LIN {X 0,Y 356.251,Z 232.015,A -85,B 0,C 180,E1 -13438.258,E2 -13438.258} C_VEL
LIN {X 0,Y 354.845,Z 225.287,A -85,B 0,C 180,E1 -13439.964,E2 -13439.964} C_VEL
LIN {X 0,Y 354.802,Z 225.258,A -85,B 0,C 180,E1 -13443.701,E2 -13443.701} C_VEL
LIN {X 0,Y 354.792,Z 225.291,A -85,B 0,C 180,E1 -13446.458,E2 -13446.458} C_VEL
LIN {X 0,Y 354.762,Z 225.285,A -85,B 0,C 180,E1 -13449.411,E2 -13449.411} C_VEL
LIN {X 0,Y 354.779,Z 225.283,A -85,B 0,C 180,E1 -13452.866,E2 -13452.866} C_VEL
LIN {X 0,Y 354.759,Z 225.293,A -85,B 0,C 180,E1 -13456.102,E2 -13456.102} C_VEL
LIN {X 0,Y 354.758,Z 225.282,A -85,B 0,C 180,E1 -13459.175,E2 -13459.175} C_VEL
LIN {X 0,Y 354.793,Z 225.285,A -85,B 0,C 180,E1 -13462.403,E2 -13462.403} C_VEL
LIN {X 0,Y 354.804,Z 225.27,A -85,B 0,C 180,E1 -13464.94,E2 -13464.94} C_VEL
LIN {X 0,Y 354.785,Z 225.285,A -85,B 0,C 180,E1 -13468.404,E2 -13468.404} C_VEL
LIN {X 0,Y 354.788,Z 225.272,A -85,B 0,C 180,E1 -13471.614,E2 -13471.614} C_VEL
LIN {X 0,Y 354.825,Z 225.275,A -85,B 0,C 180,E1 -13475.657,E2 -13475.657} C_VEL
LIN {X 0,Y 354.816,Z 225.265,A -85,B 0,C 180,E1 -13479.113,E2 -13479.113} C_VEL
LIN {X 0,Y 354.869,Z 225.279,A -85,B 0,C 180,E1 -13482.719,E2 -13482.719} C_VEL
LIN {X 0,Y 354.942,Z 225.244,A -85,B 0,C 180,E1 -13486.255,E2 -13486.255} C_VEL
LIN {X 0,Y 354.946,Z 225.269,A -85,B 0,C 180,E1 -13489.735,E2 -13489.735} C_VEL
LIN {X 0,Y 355.073,Z 225.238,A -85,B 0,C 180,E1 -13493.18,E2 -13493.18} C_VEL
LIN {X 0,Y 355.224,Z 225.23,A -85,B 0,C 180,E1 -13497.733,E2 -13497.733} C_VEL
LIN {X 0,Y 355.166,Z 225.228,A -85,B 0,C 180,E1 -13501.134,E2 -13501.134} C_VEL
LIN {X 0,Y 355.221,Z 225.21,A -85,B 0,C 180,E1 -13502.268,E2 -13502.268} C_VEL
LIN {X 0,Y 355.116,Z 225.244,A -85,B 0,C 180,E1 -13506.82,E2 -13506.82} C_VEL
LIN {X 0,Y 354.969,Z 225.243,A -85,B 0,C 180,E1 -13510.265,E2 -13510.265} C_VEL
LIN {X 0,Y 354.935,Z 225.272,A -85,B 0,C 180,E1 -13514.02,E2 -13514.02} C_VEL
LIN {X 0,Y 354.882,Z 225.262,A -85,B 0,C 180,E1 -13518.093,E2 -13518.093} C_VEL
LIN {X 0,Y 354.829,Z 225.279,A -85,B 0,C 180,E1 -13522.107,E2 -13522.107} C_VEL
LIN {X 0,Y 354.893,Z 225.278,A -85,B 0,C 180,E1 -13525.828,E2 -13525.828} C_VEL
LIN {X 0,Y 354.811,Z 225.278,A -85,B 0,C 180,E1 -13529.683,E2 -13529.683} C_VEL
LIN {X 0,Y 354.8,Z 225.28,A -85,B 0,C 180,E1 -13533.703,E2 -13533.703} C_VEL
LIN {X 0,Y 354.794,Z 225.293,A -85,B 0,C 180,E1 -13536.461,E2 -13536.461} C_VEL
LIN {X 0,Y 354.819,Z 225.288,A -85,B 0,C 180,E1 -13539.425,E2 -13539.425} C_VEL
LIN {X 0,Y 354.785,Z 225.29,A -85,B 0,C 180,E1 -13542.869,E2 -13542.869} C_VEL
LIN {X 0,Y 354.766,Z 225.294,A -85,B 0,C 180,E1 -13546.105,E2 -13546.105} C_VEL
LIN {X 0,Y 354.786,Z 225.29,A -85,B 0,C 180,E1 -13549.181,E2 -13549.181} C_VEL
LIN {X 0,Y 354.841,Z 225.283,A -85,B 0,C 180,E1 -13551.977,E2 -13551.977} C_VEL
LIN {X 0,Y 355.818,Z 228.129,A -85,B 0,C 180,E1 -13552.146,E2 -13552.146} C_VEL
LIN {X 0,Y 362.138,Z 240.848,A -85,B 0,C 180,E1 -13552.959,E2 -13552.959} C_VEL
LIN {X 0,Y 365.502,Z 249.264,A -85,B 0,C 180,E1 -13553.412,E2 -13553.412} C_VEL
LIN {X 0,Y 366.502,Z 255.255,A -85,B 0,C 180,E1 -13553.621,E2 -13553.621} C_VEL
LIN {X 0,Y 364.606,Z 337.997,A -85,B 0,C 180,E1 -13555.284,E2 -13555.284} C_VEL
LIN {X 0,Y 364.035,Z 351.449,A -85,B 0,C 180,E1 -13555.767,E2 -13555.767} C_VEL
LIN {X 0,Y 363.357,Z 362.814,A -85,B 0,C 180,E1 -13556.384,E2 -13556.384} C_VEL
LIN {X 0,Y 362.251,Z 374.947,A -85,B 0,C 180,E1 -13557.263,E2 -13557.263} C_VEL
LIN {X 0,Y 361.138,Z 385.976,A -85,B 0,C 180,E1 -13558.304,E2 -13558.304} C_VEL
LIN {X 0,Y 359.839,Z 396.022,A -85,B 0,C 180,E1 -13559.484,E2 -13559.484} C_VEL
LIN {X 0,Y 358.474,Z 406.105,A -85,B 0,C 180,E1 -13560.974,E2 -13560.974} C_VEL
LIN {X 0,Y 357.292,Z 414.918,A -85,B 0,C 180,E1 -13562.599,E2 -13562.599} C_VEL
LIN {X 0,Y 356.138,Z 422.187,A -85,B 0,C 180,E1 -13564.271,E2 -13564.271} C_VEL
LIN {X 0,Y 355.23,Z 428.414,A -85,B 0,C 180,E1 -13566.074,E2 -13566.074} C_VEL
LIN {X 0,Y 354.488,Z 433.26,A -85,B 0,C 180,E1 -13567.873,E2 -13567.873} C_VEL
LIN {X 0,Y 353.956,Z 436.89,A -85,B 0,C 180,E1 -13569.669,E2 -13569.669} C_VEL
LIN {X 0,Y 353.537,Z 439.423,A -85,B 0,C 180,E1 -13571.455,E2 -13571.455} C_VEL
LIN {X 0,Y 353.399,Z 440.56,A -85,B 0,C 180,E1 -13572.665,E2 -13572.665} C_VEL
LIN {X 0,Y 353.286,Z 441.221,A -85,B 0,C 180,E1 -13573.83,E2 -13573.83} C_VEL
LIN {X 0,Y 353.19,Z 441.496,A -85,B 0,C 180,E1 -13575.009,E2 -13575.009} C_VEL
LIN {X 0,Y 353.235,Z 440.909,A -85,B 0,C 180,E1 -13577.14,E2 -13577.14} C_VEL
LIN {X 0,Y 353.276,Z 439.77,A -85,B 0,C 180,E1 -13578.526,E2 -13578.526} C_VEL
LIN {X 0,Y 353.313,Z 438.384,A -85,B 0,C 180,E1 -13579.688,E2 -13579.688} C_VEL
LIN {X 0,Y 353.58,Z 435.443,A -85,B 0,C 180,E1 -13581.428,E2 -13581.428} C_VEL
LIN {X 0,Y 353.899,Z 431.364,A -85,B 0,C 180,E1 -13583.192,E2 -13583.192} C_VEL
LIN {X 0,Y 354.237,Z 426.314,A -85,B 0,C 180,E1 -13584.879,E2 -13584.879} C_VEL
LIN {X 0,Y 354.84,Z 419.838,A -85,B 0,C 180,E1 -13586.595,E2 -13586.595} C_VEL
LIN {X 0,Y 355.605,Z 411.8,A -85,B 0,C 180,E1 -13588.302,E2 -13588.302} C_VEL
LIN {X 0,Y 356.382,Z 403.578,A -85,B 0,C 180,E1 -13589.719,E2 -13589.719} C_VEL
LIN {X 0,Y 357.34,Z 393.444,A -85,B 0,C 180,E1 -13591.128,E2 -13591.128} C_VEL
LIN {X 0,Y 358.376,Z 382.087,A -85,B 0,C 180,E1 -13592.39,E2 -13592.39} C_VEL
LIN {X 0,Y 359.209,Z 370.828,A -85,B 0,C 180,E1 -13593.366,E2 -13593.366} C_VEL
LIN {X 0,Y 359.788,Z 359.435,A -85,B 0,C 180,E1 -13594.132,E2 -13594.132} C_VEL
LIN {X 0,Y 360.335,Z 346.612,A -85,B 0,C 180,E1 -13594.756,E2 -13594.756} C_VEL
LIN {X 0,Y 360.685,Z 334.356,A -85,B 0,C 180,E1 -13595.137,E2 -13595.137} C_VEL
LIN {X 0,Y 361.954,Z 253.14,A -85,B 0,C 180,E1 -13596.743,E2 -13596.743} C_VEL
LIN {X 0,Y 359.063,Z 236.78,A -85,B 0,C 180,E1 -13597.225,E2 -13597.225} C_VEL
LIN {X 0,Y 355.076,Z 225.258,A -85,B 0,C 180,E1 -13597.679,E2 -13597.679} C_VEL
LIN {X 0,Y 354.933,Z 225.27,A -85,B 0,C 180,E1 -13601.515,E2 -13601.515} C_VEL
LIN {X 0,Y 354.233,Z 225.363,A -85,B 0,C 180,E1 -13602.462,E2 -13602.462} C_VEL
LIN {X 0,Y 351.375,Z 225.722,A -85,B 0,C 180,E1 -13604.002,E2 -13604.002} C_VEL
LIN {X 0,Y 348.97,Z 226.024,A -85,B 0,C 180,E1 -13605.248,E2 -13605.248} C_VEL
LIN {X 0,Y 347.931,Z 226.15,A -85,B 0,C 180,E1 -13606.212,E2 -13606.212} C_VEL
LIN {X 0,Y 347.842,Z 226.158,A -85,B 0,C 180,E1 -13606.539,E2 -13606.539} C_VEL
LIN {X 0,Y 347.859,Z 226.152,A -85,B 0,C 180,E1 -13608.861,E2 -13608.861} C_VEL
LIN {X 0,Y 347.762,Z 226.165,A -85,B 0,C 180,E1 -13612.581,E2 -13612.581} C_VEL
LIN {X 0,Y 347.745,Z 226.165,A -85,B 0,C 180,E1 -13615.115,E2 -13615.115} C_VEL
LIN {X 0,Y 347.735,Z 226.169,A -85,B 0,C 180,E1 -13617.702,E2 -13617.702} C_VEL
LIN {X 0,Y 347.744,Z 226.167,A -85,B 0,C 180,E1 -13620.35,E2 -13620.35} C_VEL
LIN {X 0,Y 347.754,Z 226.168,A -85,B 0,C 180,E1 -13624.044,E2 -13624.044} C_VEL
LIN {X 0,Y 347.76,Z 226.166,A -85,B 0,C 180,E1 -13627.322,E2 -13627.322} C_VEL
LIN {X 0,Y 347.702,Z 226.171,A -85,B 0,C 180,E1 -13630.303,E2 -13630.303} C_VEL
LIN {X 0,Y 347.727,Z 226.173,A -85,B 0,C 180,E1 -13633.409,E2 -13633.409} C_VEL
LIN {X 0,Y 347.728,Z 226.168,A -85,B 0,C 180,E1 -13636.687,E2 -13636.687} C_VEL
LIN {X 0,Y 347.707,Z 226.17,A -85,B 0,C 180,E1 -13640.183,E2 -13640.183} C_VEL
LIN {X 0,Y 347.759,Z 226.165,A -85,B 0,C 180,E1 -13642.678,E2 -13642.678} C_VEL
LIN {X 0,Y 347.754,Z 226.164,A -85,B 0,C 180,E1 -13645.957,E2 -13645.957} C_VEL
LIN {X 0,Y 347.735,Z 226.167,A -85,B 0,C 180,E1 -13649.65,E2 -13649.65} C_VEL
LIN {X 0,Y 347.739,Z 226.166,A -85,B 0,C 180,E1 -13653.6,E2 -13653.6} C_VEL
LIN {X 0,Y 347.835,Z 226.225,A -85,B 0,C 180,E1 -13656.362,E2 -13656.362} C_VEL
LIN {X 0,Y 348.763,Z 231.232,A -85,B 0,C 180,E1 -13657.799,E2 -13657.799} C_VEL
LIN {X 0,Y 352.134,Z 244.583,A -85,B 0,C 180,E1 -13658.321,E2 -13658.321} C_VEL
LIN {X 0,Y 354.029,Z 256.193,A -85,B 0,C 180,E1 -13658.724,E2 -13658.724} C_VEL
LIN {X 0,Y 351.664,Z 339.815,A -85,B 0,C 180,E1 -13661.049,E2 -13661.049} C_VEL
LIN {X 0,Y 351.252,Z 352.875,A -85,B 0,C 180,E1 -13661.631,E2 -13661.631} C_VEL
LIN {X 0,Y 350.773,Z 364.722,A -85,B 0,C 180,E1 -13662.359,E2 -13662.359} C_VEL
LIN {X 0,Y 350.003,Z 377.261,A -85,B 0,C 180,E1 -13663.373,E2 -13663.373} C_VEL
LIN {X 0,Y 349.34,Z 388.67,A -85,B 0,C 180,E1 -13664.54,E2 -13664.54} C_VEL
LIN {X 0,Y 348.739,Z 398.714,A -85,B 0,C 180,E1 -13665.812,E2 -13665.812} C_VEL
LIN {X 0,Y 347.973,Z 409.252,A -85,B 0,C 180,E1 -13667.46,E2 -13667.46} C_VEL
LIN {X 0,Y 347.426,Z 416.873,A -85,B 0,C 180,E1 -13668.92,E2 -13668.92} C_VEL
LIN {X 0,Y 346.971,Z 424.322,A -85,B 0,C 180,E1 -13670.674,E2 -13670.674} C_VEL
LIN {X 0,Y 346.661,Z 430.262,A -85,B 0,C 180,E1 -13672.427,E2 -13672.427} C_VEL
LIN {X 0,Y 346.447,Z 434.904,A -85,B 0,C 180,E1 -13674.178,E2 -13674.178} C_VEL
LIN {X 0,Y 346.413,Z 437.37,A -85,B 0,C 180,E1 -13675.345,E2 -13675.345} C_VEL
LIN {X 0,Y 346.311,Z 439.316,A -85,B 0,C 180,E1 -13676.509,E2 -13676.509} C_VEL
LIN {X 0,Y 346.269,Z 440.807,A -85,B 0,C 180,E1 -13677.673,E2 -13677.673} C_VEL
LIN {X 0,Y 346.287,Z 441.878,A -85,B 0,C 180,E1 -13678.837,E2 -13678.837} C_VEL
LIN {X 0,Y 346.363,Z 442.493,A -85,B 0,C 180,E1 -13680,E2 -13680} C_VEL
LIN {X 0,Y 346.448,Z 442.658,A -85,B 0,C 180,E1 -13681.162,E2 -13681.162} C_VEL
LIN {X 0,Y 346.594,Z 442.409,A -85,B 0,C 180,E1 -13682.324,E2 -13682.324} C_VEL
LIN {X 0,Y 346.839,Z 441.74,A -85,B 0,C 180,E1 -13683.485,E2 -13683.485} C_VEL
LIN {X 0,Y 347.127,Z 440.595,A -85,B 0,C 180,E1 -13684.645,E2 -13684.645} C_VEL
LIN {X 0,Y 347.389,Z 439.033,A -85,B 0,C 180,E1 -13685.805,E2 -13685.805} C_VEL
LIN {X 0,Y 347.739,Z 435.862,A -85,B 0,C 180,E1 -13687.548,E2 -13687.548} C_VEL
LIN {X 0,Y 348.683,Z 431.532,A -85,B 0,C 180,E1 -13689.279,E2 -13689.279} C_VEL
LIN {X 0,Y 349.695,Z 426.024,A -85,B 0,C 180,E1 -13691.007,E2 -13691.007} C_VEL
LIN {X 0,Y 350.946,Z 419.105,A -85,B 0,C 180,E1 -13692.726,E2 -13692.726} C_VEL
LIN {X 0,Y 352.377,Z 410.495,A -85,B 0,C 180,E1 -13694.436,E2 -13694.436} C_VEL
LIN {X 0,Y 353.774,Z 401.716,A -85,B 0,C 180,E1 -13695.852,E2 -13695.852} C_VEL
LIN {X 0,Y 355.287,Z 392.173,A -85,B 0,C 180,E1 -13697.112,E2 -13697.112} C_VEL
LIN {X 0,Y 356.87,Z 380.356,A -85,B 0,C 180,E1 -13698.366,E2 -13698.366} C_VEL
LIN {X 0,Y 358.269,Z 368.264,A -85,B 0,C 180,E1 -13699.385,E2 -13699.385} C_VEL
LIN {X 0,Y 359.456,Z 355.545,A -85,B 0,C 180,E1 -13700.199,E2 -13700.199} C_VEL
LIN {X 0,Y 360.443,Z 342.476,A -85,B 0,C 180,E1 -13700.808,E2 -13700.808} C_VEL
LIN {X 0,Y 365.61,Z 264.741,A -85,B 0,C 180,E1 -13703.325,E2 -13703.325} C_VEL
LIN {X 0,Y 360.549,Z 254.309,A -85,B 0,C 180,E1 -13704.498,E2 -13704.498} C_VEL
LIN {X 0,Y 355.99,Z 246.255,A -85,B 0,C 180,E1 -13705.601,E2 -13705.601} C_VEL
LIN {X 0,Y 353.684,Z 242.531,A -85,B 0,C 180,E1 -13706.18,E2 -13706.18} C_VEL
LIN {X 0,Y 351.411,Z 238.71,A -85,B 0,C 180,E1 -13706.823,E2 -13706.823} C_VEL
LIN {X 0,Y 350.201,Z 234.367,A -85,B 0,C 180,E1 -13709.451,E2 -13709.451} C_VEL
LIN {X 0,Y 349.089,Z 230.517,A -85,B 0,C 180,E1 -13712.266,E2 -13712.266} C_VEL
LIN {X 0,Y 348.394,Z 228.278,A -85,B 0,C 180,E1 -13714.391,E2 -13714.391} C_VEL
LIN {X 0,Y 347.767,Z 226.166,A -85,B 0,C 180,E1 -13717.32,E2 -13717.32} C_VEL
LIN {X 0,Y 347.738,Z 226.169,A -85,B 0,C 180,E1 -13720.296,E2 -13720.296} C_VEL
LIN {X 0,Y 347.728,Z 226.171,A -85,B 0,C 180,E1 -13723.407,E2 -13723.407} C_VEL
LIN {X 0,Y 347.752,Z 226.314,A -85,B 0,C 180,E1 -13726.195,E2 -13726.195} C_VEL
LIN {X 0,Y 348.798,Z 229.584,A -85,B 0,C 180,E1 -13729.85,E2 -13729.85} C_VEL
LIN {X 0,Y 350.274,Z 233.844,A -85,B 0,C 180,E1 -13732.99,E2 -13732.99} C_VEL
LIN {X 0,Y 351.793,Z 239.339,A -85,B 0,C 180,E1 -13735.986,E2 -13735.986} C_VEL
LIN {X 0,Y 353.435,Z 245.803,A -85,B 0,C 180,E1 -13738.867,E2 -13738.867} C_VEL
LIN {X 0,Y 354.935,Z 253.192,A -85,B 0,C 180,E1 -13741.625,E2 -13741.625} C_VEL
LIN {X 0,Y 355.556,Z 257.298,A -85,B 0,C 180,E1 -13742.948,E2 -13742.948} C_VEL
LIN {X 0,Y 358.827,Z 269.875,A -85,B 0,C 180,E1 -13744.041,E2 -13744.041} C_VEL
LIN {X 0,Y 361.713,Z 284.255,A -85,B 0,C 180,E1 -13745.081,E2 -13745.081} C_VEL
LIN {X 0,Y 363.46,Z 296.855,A -85,B 0,C 180,E1 -13745.836,E2 -13745.836} C_VEL
LIN {X 0,Y 363.714,Z 302.155,A -85,B 0,C 180,E1 -13746.084,E2 -13746.084} C_VEL
LIN {X 0,Y 359.353,Z 371.007,A -85,B 0,C 180,E1 -13748.298,E2 -13748.298} C_VEL
LIN {X 0,Y 357.977,Z 384.376,A -85,B 0,C 180,E1 -13748.928,E2 -13748.928} C_VEL
LIN {X 0,Y 356.409,Z 397.778,A -85,B 0,C 180,E1 -13749.812,E2 -13749.812} C_VEL
LIN {X 0,Y 354.89,Z 409.166,A -85,B 0,C 180,E1 -13750.777,E2 -13750.777} C_VEL
LIN {X 0,Y 353.186,Z 420.885,A -85,B 0,C 180,E1 -13752.034,E2 -13752.034} C_VEL
LIN {X 0,Y 351.549,Z 431.561,A -85,B 0,C 180,E1 -13753.447,E2 -13753.447} C_VEL
LIN {X 0,Y 350.091,Z 440.352,A -85,B 0,C 180,E1 -13754.871,E2 -13754.871} C_VEL
LIN {X 0,Y 348.869,Z 449.007,A -85,B 0,C 180,E1 -13756.603,E2 -13756.603} C_VEL
LIN {X 0,Y 347.722,Z 456.072,A -85,B 0,C 180,E1 -13758.338,E2 -13758.338} C_VEL
LIN {X 0,Y 347.002,Z 461.759,A -85,B 0,C 180,E1 -13760.086,E2 -13760.086} C_VEL
LIN {X 0,Y 346.55,Z 466.231,A -85,B 0,C 180,E1 -13761.838,E2 -13761.838} C_VEL
LIN {X 0,Y 346.327,Z 468.587,A -85,B 0,C 180,E1 -13763.005,E2 -13763.005} C_VEL
LIN {X 0,Y 346.201,Z 470.469,A -85,B 0,C 180,E1 -13764.173,E2 -13764.173} C_VEL
LIN {X 0,Y 346.171,Z 471.923,A -85,B 0,C 180,E1 -13765.341,E2 -13765.341} C_VEL
LIN {X 0,Y 346.164,Z 472.937,A -85,B 0,C 180,E1 -13766.507,E2 -13766.507} C_VEL
LIN {X 0,Y 346.159,Z 473.475,A -85,B 0,C 180,E1 -13767.672,E2 -13767.672} C_VEL
LIN {X 0,Y 346.29,Z 473.596,A -85,B 0,C 180,E1 -13768.836,E2 -13768.836} C_VEL
LIN {X 0,Y 346.361,Z 473.287,A -85,B 0,C 180,E1 -13769.999,E2 -13769.999} C_VEL
LIN {X 0,Y 346.375,Z 472.501,A -85,B 0,C 180,E1 -13771.161,E2 -13771.161} C_VEL
LIN {X 0,Y 346.207,Z 471.307,A -85,B 0,C 180,E1 -13773.49,E2 -13773.49} C_VEL
LIN {X 0,Y 346.214,Z 470.177,A -85,B 0,C 180,E1 -13774.656,E2 -13774.656} C_VEL
LIN {X 0,Y 346.241,Z 468.394,A -85,B 0,C 180,E1 -13775.955,E2 -13775.955} C_VEL
LIN {X 0,Y 346.508,Z 464.183,A -85,B 0,C 180,E1 -13778.161,E2 -13778.161} C_VEL
LIN {X 0,Y 346.935,Z 459.588,A -85,B 0,C 180,E1 -13779.914,E2 -13779.914} C_VEL
LIN {X 0,Y 347.737,Z 452.634,A -85,B 0,C 180,E1 -13781.955,E2 -13781.955} C_VEL
LIN {X 0,Y 348.863,Z 445.128,A -85,B 0,C 180,E1 -13783.691,E2 -13783.691} C_VEL
LIN {X 0,Y 349.803,Z 437.474,A -85,B 0,C 180,E1 -13785.139,E2 -13785.139} C_VEL
LIN {X 0,Y 351.157,Z 428.129,A -85,B 0,C 180,E1 -13786.569,E2 -13786.569} C_VEL
LIN {X 0,Y 352.603,Z 417.768,A -85,B 0,C 180,E1 -13787.844,E2 -13787.844} C_VEL
LIN {X 0,Y 354.075,Z 406.259,A -85,B 0,C 180,E1 -13788.966,E2 -13788.966} C_VEL
LIN {X 0,Y 355.281,Z 394.013,A -85,B 0,C 180,E1 -13789.875,E2 -13789.875} C_VEL
LIN {X 0,Y 356.446,Z 381.138,A -85,B 0,C 180,E1 -13790.56,E2 -13790.56} C_VEL
LIN {X 0,Y 357.191,Z 368.068,A -85,B 0,C 180,E1 -13791.014,E2 -13791.014} C_VEL
LIN {X 0,Y 358.566,Z 299.255,A -85,B 0,C 180,E1 -13792.452,E2 -13792.452} C_VEL
LIN {X 0,Y 356.048,Z 280.739,A -85,B 0,C 180,E1 -13793.066,E2 -13793.066} C_VEL
LIN {X 0,Y 350.747,Z 250.28,A -85,B 0,C 180,E1 -13794.222,E2 -13794.222} C_VEL
LIN {X 0,Y 351.283,Z 245.173,A -85,B 0,C 180,E1 -13795.395,E2 -13795.395} C_VEL
LIN {X 0,Y 350.496,Z 239.332,A -85,B 0,C 180,E1 -13796.817,E2 -13796.817} C_VEL
LIN {X 0,Y 347.82,Z 226.162,A -85,B 0,C 180,E1 -13800.162,E2 -13800.162} C_VEL
LIN {X 0,Y 347.74,Z 226.141,A -85,B 0,C 180,E1 -13804.463,E2 -13804.463} C_VEL
LIN {X 0,Y 347.757,Z 226.162,A -85,B 0,C 180,E1 -13807.985,E2 -13807.985} C_VEL
LIN {X 0,Y 347.738,Z 226.166,A -85,B 0,C 180,E1 -13811.83,E2 -13811.83} C_VEL
LIN {X 0,Y 347.699,Z 226.171,A -85,B 0,C 180,E1 -13815.026,E2 -13815.026} C_VEL
LIN {X 0,Y 347.734,Z 226.153,A -85,B 0,C 180,E1 -13818.398,E2 -13818.398} C_VEL
LIN {X 0,Y 347.749,Z 226.161,A -85,B 0,C 180,E1 -13822.678,E2 -13822.678} C_VEL
LIN {X 0,Y 347.741,Z 226.162,A -85,B 0,C 180,E1 -13825.955,E2 -13825.955} C_VEL
LIN {X 0,Y 347.732,Z 226.15,A -85,B 0,C 180,E1 -13829.651,E2 -13829.651} C_VEL
LIN {X 0,Y 347.731,Z 226.165,A -85,B 0,C 180,E1 -13833.6,E2 -13833.6} C_VEL
LIN {X 0,Y 347.753,Z 226.156,A -85,B 0,C 180,E1 -13836.159,E2 -13836.159} C_VEL
LIN {X 0,Y 347.789,Z 226.15,A -85,B 0,C 180,E1 -13839.908,E2 -13839.908} C_VEL
LIN {X 0,Y 347.82,Z 226.15,A -85,B 0,C 180,E1 -13843.568,E2 -13843.568} C_VEL
LIN {X 0,Y 347.88,Z 226.13,A -85,B 0,C 180,E1 -13847.16,E2 -13847.16} C_VEL
LIN {X 0,Y 347.926,Z 226.146,A -85,B 0,C 180,E1 -13850.701,E2 -13850.701} C_VEL
LIN {X 0,Y 348.026,Z 226.106,A -85,B 0,C 180,E1 -13854.205,E2 -13854.205} C_VEL
LIN {X 0,Y 348.185,Z 226.106,A -85,B 0,C 180,E1 -13857.687,E2 -13857.687} C_VEL
LIN {X 0,Y 348.134,Z 226.104,A -85,B 0,C 180,E1 -13861.157,E2 -13861.157} C_VEL
LIN {X 0,Y 348.182,Z 226.085,A -85,B 0,C 180,E1 -13862.314,E2 -13862.314} C_VEL
LIN {X 0,Y 348.082,Z 226.12,A -85,B 0,C 180,E1 -13866.958,E2 -13866.958} C_VEL
LIN {X 0,Y 347.92,Z 226.12,A -85,B 0,C 180,E1 -13870.475,E2 -13870.475} C_VEL
LIN {X 0,Y 347.891,Z 226.148,A -85,B 0,C 180,E1 -13874.151,E2 -13874.151} C_VEL
LIN {X 0,Y 347.821,Z 226.143,A -85,B 0,C 180,E1 -13878.26,E2 -13878.26} C_VEL
LIN {X 0,Y 347.783,Z 226.161,A -85,B 0,C 180,E1 -13881.637,E2 -13881.637} C_VEL
LIN {X 0,Y 347.805,Z 226.152,A -85,B 0,C 180,E1 -13885.109,E2 -13885.109} C_VEL
LIN {X 0,Y 347.802,Z 226.157,A -85,B 0,C 180,E1 -13887.695,E2 -13887.695} C_VEL
LIN {X 0,Y 347.743,Z 226.164,A -85,B 0,C 180,E1 -13890.349,E2 -13890.349} C_VEL
LIN {X 0,Y 347.743,Z 226.158,A -85,B 0,C 180,E1 -13894.045,E2 -13894.045} C_VEL
LIN {X 0,Y 347.758,Z 226.165,A -85,B 0,C 180,E1 -13897.322,E2 -13897.322} C_VEL
LIN {X 0,Y 347.729,Z 226.173,A -85,B 0,C 180,E1 -13900.298,E2 -13900.298} C_VEL
LIN {X 0,Y 347.72,Z 226.174,A -85,B 0,C 180,E1 -13903.409,E2 -13903.409} C_VEL
LIN {X 0,Y 347.722,Z 226.172,A -85,B 0,C 180,E1 -13906.688,E2 -13906.688} C_VEL
LIN {X 0,Y 347.745,Z 226.166,A -85,B 0,C 180,E1 -13910.175,E2 -13910.175} C_VEL
LIN {X 0,Y 347.795,Z 226.161,A -85,B 0,C 180,E1 -13911.375,E2 -13911.375} C_VEL
LIN {X 0,Y 348.88,Z 229.117,A -85,B 0,C 180,E1 -13911.557,E2 -13911.557} C_VEL
LIN {X 0,Y 355.974,Z 243.175,A -85,B 0,C 180,E1 -13912.5,E2 -13912.5} C_VEL
LIN {X 0,Y 359.435,Z 251.984,A -85,B 0,C 180,E1 -13912.984,E2 -13912.984} C_VEL
LIN {X 0,Y 360.147,Z 256.344,A -85,B 0,C 180,E1 -13913.139,E2 -13913.139} C_VEL
LIN {X 0,Y 358.158,Z 338.002,A -85,B 0,C 180,E1 -13914.803,E2 -13914.803} C_VEL
LIN {X 0,Y 357.6,Z 351.228,A -85,B 0,C 180,E1 -13915.28,E2 -13915.28} C_VEL
LIN {X 0,Y 356.917,Z 362.189,A -85,B 0,C 180,E1 -13915.869,E2 -13915.869} C_VEL
LIN {X 0,Y 355.784,Z 374.511,A -85,B 0,C 180,E1 -13916.761,E2 -13916.761} C_VEL
LIN {X 0,Y 354.625,Z 385.685,A -85,B 0,C 180,E1 -13917.82,E2 -13917.82} C_VEL
LIN {X 0,Y 353.253,Z 395.856,A -85,B 0,C 180,E1 -13919.019,E2 -13919.019} C_VEL
LIN {X 0,Y 351.934,Z 405.115,A -85,B 0,C 180,E1 -13920.381,E2 -13920.381} C_VEL
LIN {X 0,Y 350.783,Z 413.135,A -85,B 0,C 180,E1 -13921.831,E2 -13921.831} C_VEL
LIN {X 0,Y 349.622,Z 420.41,A -85,B 0,C 180,E1 -13923.433,E2 -13923.433} C_VEL
LIN {X 0,Y 348.634,Z 426.591,A -85,B 0,C 180,E1 -13925.115,E2 -13925.115} C_VEL
LIN {X 0,Y 347.846,Z 431.539,A -85,B 0,C 180,E1 -13926.799,E2 -13926.799} C_VEL
LIN {X 0,Y 347.195,Z 435.707,A -85,B 0,C 180,E1 -13928.633,E2 -13928.633} C_VEL
LIN {X 0,Y 346.833,Z 437.83,A -85,B 0,C 180,E1 -13929.852,E2 -13929.852} C_VEL
LIN {X 0,Y 346.532,Z 439.477,A -85,B 0,C 180,E1 -13931.066,E2 -13931.066} C_VEL
LIN {X 0,Y 346.334,Z 440.868,A -85,B 0,C 180,E1 -13932.508,E2 -13932.508} C_VEL
LIN {X 0,Y 346.11,Z 441.786,A -85,B 0,C 180,E1 -13934.695,E2 -13934.695} C_VEL
LIN {X 0,Y 346.076,Z 441.72,A -85,B 0,C 180,E1 -13935.897,E2 -13935.897} C_VEL
LIN {X 0,Y 346.136,Z 441.22,A -85,B 0,C 180,E1 -13937.096,E2 -13937.096} C_VEL
LIN {X 0,Y 346.166,Z 440.291,A -85,B 0,C 180,E1 -13938.288,E2 -13938.288} C_VEL
LIN {X 0,Y 346.203,Z 438.968,A -85,B 0,C 180,E1 -13939.474,E2 -13939.474} C_VEL
LIN {X 0,Y 346.454,Z 436.147,A -85,B 0,C 180,E1 -13941.25,E2 -13941.25} C_VEL
LIN {X 0,Y 346.819,Z 431.855,A -85,B 0,C 180,E1 -13943.195,E2 -13943.195} C_VEL
LIN {X 0,Y 347.129,Z 427.318,A -85,B 0,C 180,E1 -13944.774,E2 -13944.774} C_VEL
LIN {X 0,Y 347.739,Z 421.016,A -85,B 0,C 180,E1 -13946.525,E2 -13946.525} C_VEL
LIN {X 0,Y 348.485,Z 413.157,A -85,B 0,C 180,E1 -13948.268,E2 -13948.268} C_VEL
LIN {X 0,Y 349.287,Z 405.14,A -85,B 0,C 180,E1 -13949.713,E2 -13949.713} C_VEL
LIN {X 0,Y 350.251,Z 395.376,A -85,B 0,C 180,E1 -13951.151,E2 -13951.151} C_VEL
LIN {X 0,Y 351.314,Z 384.221,A -85,B 0,C 180,E1 -13952.452,E2 -13952.452} C_VEL
LIN {X 0,Y 352.283,Z 372.062,A -85,B 0,C 180,E1 -13953.566,E2 -13953.566} C_VEL
LIN {X 0,Y 352.928,Z 359.939,A -85,B 0,C 180,E1 -13954.405,E2 -13954.405} C_VEL
LIN {X 0,Y 353.517,Z 346.676,A -85,B 0,C 180,E1 -13955.062,E2 -13955.062} C_VEL
LIN {X 0,Y 353.863,Z 334.204,A -85,B 0,C 180,E1 -13955.45,E2 -13955.45} C_VEL
LIN {X 0,Y 355.189,Z 254.031,A -85,B 0,C 180,E1 -13957.064,E2 -13957.064} C_VEL
LIN {X 0,Y 352.559,Z 238.973,A -85,B 0,C 180,E1 -13957.517,E2 -13957.517} C_VEL
LIN {X 0,Y 348.023,Z 226.135,A -85,B 0,C 180,E1 -13958.049,E2 -13958.049} C_VEL
LIN {X 0,Y 347.889,Z 226.147,A -85,B 0,C 180,E1 -13961.656,E2 -13961.656} C_VEL
LIN {X 0,Y 347.872,Z 226.15,A -85,B 0,C 180,E1 -13965.228,E2 -13965.228} C_VEL
LIN {X 0,Y 347.842,Z 226.158,A -85,B 0,C 180,E1 -13966.539,E2 -13966.539} C_VEL
LIN {X 0,Y 347.148,Z 226.241,A -85,B 0,C 180,E1 -13967.505,E2 -13967.505} C_VEL
LIN {X 0,Y 344.244,Z 226.602,A -85,B 0,C 180,E1 -13969.075,E2 -13969.075} C_VEL
LIN {X 0,Y 341.811,Z 226.91,A -85,B 0,C 180,E1 -13970.346,E2 -13970.346} C_VEL
LIN {X 0,Y 340.792,Z 227.032,A -85,B 0,C 180,E1 -13971.331,E2 -13971.331} C_VEL
LIN {X 0,Y 340.723,Z 227.041,A -85,B 0,C 180,E1 -13971.664,E2 -13971.664} C_VEL
LIN {X 0,Y 340.714,Z 227.042,A -85,B 0,C 180,E1 -13974.823,E2 -13974.823} C_VEL
LIN {X 0,Y 340.685,Z 227.047,A -85,B 0,C 180,E1 -13978.326,E2 -13978.326} C_VEL
LIN {X 0,Y 340.7,Z 227.043,A -85,B 0,C 180,E1 -13981.046,E2 -13981.046} C_VEL
LIN {X 0,Y 340.722,Z 227.042,A -85,B 0,C 180,E1 -13985.28,E2 -13985.28} C_VEL
LIN {X 0,Y 340.699,Z 227.043,A -85,B 0,C 180,E1 -13988.383,E2 -13988.383} C_VEL
LIN {X 0,Y 340.696,Z 227.044,A -85,B 0,C 180,E1 -13992.044,E2 -13992.044} C_VEL
LIN {X 0,Y 340.655,Z 227.048,A -85,B 0,C 180,E1 -13996.228,E2 -13996.228} C_VEL
LIN {X 0,Y 340.674,Z 227.047,A -85,B 0,C 180,E1 -13998.688,E2 -13998.688} C_VEL
LIN {X 0,Y 340.723,Z 227.041,A -85,B 0,C 180,E1 -14001.771,E2 -14001.771} C_VEL
LIN {X 0,Y 340.728,Z 227.041,A -85,B 0,C 180,E1 -14005.596,E2 -14005.596} C_VEL
LIN {X 0,Y 340.688,Z 227.05,A -85,B 0,C 180,E1 -14008.954,E2 -14008.954} C_VEL
LIN {X 0,Y 340.692,Z 227.046,A -85,B 0,C 180,E1 -14012.505,E2 -14012.505} C_VEL
LIN {X 0,Y 340.784,Z 227.049,A -85,B 0,C 180,E1 -14016.206,E2 -14016.206} C_VEL
LIN {X 0,Y 341.6,Z 231.537,A -85,B 0,C 180,E1 -14017.512,E2 -14017.512} C_VEL
LIN {X 0,Y 345.32,Z 245.986,A -85,B 0,C 180,E1 -14018.096,E2 -14018.096} C_VEL
LIN {X 0,Y 347.119,Z 256.377,A -85,B 0,C 180,E1 -14018.472,E2 -14018.472} C_VEL
LIN {X 0,Y 344.644,Z 340.237,A -85,B 0,C 180,E1 -14020.88,E2 -14020.88} C_VEL
LIN {X 0,Y 344.191,Z 354.626,A -85,B 0,C 180,E1 -14021.549,E2 -14021.549} C_VEL
LIN {X 0,Y 343.598,Z 367.998,A -85,B 0,C 180,E1 -14022.44,E2 -14022.44} C_VEL
LIN {X 0,Y 342.83,Z 379.972,A -85,B 0,C 180,E1 -14023.474,E2 -14023.474} C_VEL
LIN {X 0,Y 342.061,Z 391.134,A -85,B 0,C 180,E1 -14024.698,E2 -14024.698} C_VEL
LIN {X 0,Y 341.557,Z 400.868,A -85,B 0,C 180,E1 -14026.008,E2 -14026.008} C_VEL
LIN {X 0,Y 340.845,Z 410.007,A -85,B 0,C 180,E1 -14027.496,E2 -14027.496} C_VEL
LIN {X 0,Y 340.245,Z 418.883,A -85,B 0,C 180,E1 -14029.286,E2 -14029.286} C_VEL
LIN {X 0,Y 339.795,Z 426.015,A -85,B 0,C 180,E1 -14031.076,E2 -14031.076} C_VEL
LIN {X 0,Y 339.485,Z 431.702,A -85,B 0,C 180,E1 -14032.864,E2 -14032.864} C_VEL
LIN {X 0,Y 339.326,Z 436.112,A -85,B 0,C 180,E1 -14034.652,E2 -14034.652} C_VEL
LIN {X 0,Y 339.234,Z 439.371,A -85,B 0,C 180,E1 -14036.436,E2 -14036.436} C_VEL
LIN {X 0,Y 339.176,Z 440.937,A -85,B 0,C 180,E1 -14037.625,E2 -14037.625} C_VEL
LIN {X 0,Y 339.19,Z 442.074,A -85,B 0,C 180,E1 -14038.812,E2 -14038.812} C_VEL
LIN {X 0,Y 339.268,Z 442.796,A -85,B 0,C 180,E1 -14040,E2 -14040} C_VEL
LIN {X 0,Y 339.389,Z 443.05,A -85,B 0,C 180,E1 -14041.186,E2 -14041.186} C_VEL
LIN {X 0,Y 339.543,Z 442.868,A -85,B 0,C 180,E1 -14042.372,E2 -14042.372} C_VEL
LIN {X 0,Y 339.799,Z 442.274,A -85,B 0,C 180,E1 -14043.557,E2 -14043.557} C_VEL
LIN {X 0,Y 340.1,Z 441.253,A -85,B 0,C 180,E1 -14044.741,E2 -14044.741} C_VEL
LIN {X 0,Y 340.369,Z 439.762,A -85,B 0,C 180,E1 -14045.926,E2 -14045.926} C_VEL
LIN {X 0,Y 340.756,Z 436.736,A -85,B 0,C 180,E1 -14047.704,E2 -14047.704} C_VEL
LIN {X 0,Y 341.753,Z 432.563,A -85,B 0,C 180,E1 -14049.469,E2 -14049.469} C_VEL
LIN {X 0,Y 343.063,Z 426.214,A -85,B 0,C 180,E1 -14051.521,E2 -14051.521} C_VEL
LIN {X 0,Y 344.385,Z 419.252,A -85,B 0,C 180,E1 -14053.272,E2 -14053.272} C_VEL
LIN {X 0,Y 345.958,Z 410.61,A -85,B 0,C 180,E1 -14055.011,E2 -14055.011} C_VEL
LIN {X 0,Y 347.687,Z 400.817,A -85,B 0,C 180,E1 -14056.59,E2 -14056.59} C_VEL
LIN {X 0,Y 349.471,Z 389.781,A -85,B 0,C 180,E1 -14058.011,E2 -14058.011} C_VEL
LIN {X 0,Y 350.97,Z 379.08,A -85,B 0,C 180,E1 -14059.125,E2 -14059.125} C_VEL
LIN {X 0,Y 352.486,Z 366.829,A -85,B 0,C 180,E1 -14060.128,E2 -14060.128} C_VEL
LIN {X 0,Y 353.76,Z 353.226,A -85,B 0,C 180,E1 -14060.983,E2 -14060.983} C_VEL
LIN {X 0,Y 354.887,Z 337.752,A -85,B 0,C 180,E1 -14061.643,E2 -14061.643} C_VEL
LIN {X 0,Y 360.039,Z 267.819,A -85,B 0,C 180,E1 -14063.955,E2 -14063.955} C_VEL
LIN {X 0,Y 359.7,Z 266.468,A -85,B 0,C 180,E1 -14064.066,E2 -14064.066} C_VEL
LIN {X 0,Y 354.327,Z 255.635,A -85,B 0,C 180,E1 -14065.405,E2 -14065.405} C_VEL
LIN {X 0,Y 349.549,Z 247.582,A -85,B 0,C 180,E1 -14066.657,E2 -14066.657} C_VEL
LIN {X 0,Y 346.812,Z 243.405,A -85,B 0,C 180,E1 -14067.412,E2 -14067.412} C_VEL
LIN {X 0,Y 344.489,Z 239.643,A -85,B 0,C 180,E1 -14068.115,E2 -14068.115} C_VEL
LIN {X 0,Y 343.375,Z 235.771,A -85,B 0,C 180,E1 -14070.776,E2 -14070.776} C_VEL
LIN {X 0,Y 342.404,Z 232.42,A -85,B 0,C 180,E1 -14073.655,E2 -14073.655} C_VEL
LIN {X 0,Y 341.674,Z 230.014,A -85,B 0,C 180,E1 -14076.657,E2 -14076.657} C_VEL
LIN {X 0,Y 341.159,Z 228.768,A -85,B 0,C 180,E1 -14079.688,E2 -14079.688} C_VEL
LIN {X 0,Y 341.091,Z 228.68,A -85,B 0,C 180,E1 -14082.839,E2 -14082.839} C_VEL
LIN {X 0,Y 341.647,Z 229.85,A -85,B 0,C 180,E1 -14086.053,E2 -14086.053} C_VEL
LIN {X 0,Y 342.47,Z 232.706,A -85,B 0,C 180,E1 -14089.402,E2 -14089.402} C_VEL
LIN {X 0,Y 343.978,Z 237.078,A -85,B 0,C 180,E1 -14092.828,E2 -14092.828} C_VEL
LIN {X 0,Y 345.531,Z 242.679,A -85,B 0,C 180,E1 -14095.989,E2 -14095.989} C_VEL
LIN {X 0,Y 347.218,Z 249.706,A -85,B 0,C 180,E1 -14099.158,E2 -14099.158} C_VEL
LIN {X 0,Y 348.502,Z 256.425,A -85,B 0,C 180,E1 -14101.693,E2 -14101.693} C_VEL
LIN {X 0,Y 350.746,Z 261.246,A -85,B 0,C 180,E1 -14102.347,E2 -14102.347} C_VEL
LIN {X 0,Y 353.132,Z 270.252,A -85,B 0,C 180,E1 -14103.193,E2 -14103.193} C_VEL
LIN {X 0,Y 355.865,Z 283.758,A -85,B 0,C 180,E1 -14104.247,E2 -14104.247} C_VEL
LIN {X 0,Y 357.73,Z 296.729,A -85,B 0,C 180,E1 -14105.09,E2 -14105.09} C_VEL
LIN {X 0,Y 358.082,Z 303.505,A -85,B 0,C 180,E1 -14105.43,E2 -14105.43} C_VEL
LIN {X 0,Y 353.463,Z 370.44,A -85,B 0,C 180,E1 -14107.649,E2 -14107.649} C_VEL
LIN {X 0,Y 351.955,Z 384.282,A -85,B 0,C 180,E1 -14108.319,E2 -14108.319} C_VEL
LIN {X 0,Y 350.146,Z 398.443,A -85,B 0,C 180,E1 -14109.281,E2 -14109.281} C_VEL
LIN {X 0,Y 348.307,Z 410.903,A -85,B 0,C 180,E1 -14110.399,E2 -14110.399} C_VEL
LIN {X 0,Y 346.332,Z 423.358,A -85,B 0,C 180,E1 -14111.819,E2 -14111.819} C_VEL
LIN {X 0,Y 344.506,Z 434.331,A -85,B 0,C 180,E1 -14113.404,E2 -14113.404} C_VEL
LIN {X 0,Y 343.024,Z 442.595,A -85,B 0,C 180,E1 -14114.856,E2 -14114.856} C_VEL
LIN {X 0,Y 341.743,Z 450.759,A -85,B 0,C 180,E1 -14116.622,E2 -14116.622} C_VEL
LIN {X 0,Y 340.758,Z 456.402,A -85,B 0,C 180,E1 -14118.096,E2 -14118.096} C_VEL
LIN {X 0,Y 339.999,Z 461.92,A -85,B 0,C 180,E1 -14119.879,E2 -14119.879} C_VEL
LIN {X 0,Y 339.512,Z 466.26,A -85,B 0,C 180,E1 -14121.667,E2 -14121.667} C_VEL
LIN {X 0,Y 339.258,Z 468.523,A -85,B 0,C 180,E1 -14122.859,E2 -14122.859} C_VEL
LIN {X 0,Y 339.133,Z 470.437,A -85,B 0,C 180,E1 -14124.113,E2 -14124.113} C_VEL
LIN {X 0,Y 339.072,Z 471.742,A -85,B 0,C 180,E1 -14125.243,E2 -14125.243} C_VEL
LIN {X 0,Y 339.086,Z 472.655,A -85,B 0,C 180,E1 -14126.434,E2 -14126.434} C_VEL
LIN {X 0,Y 339.068,Z 473.14,A -85,B 0,C 180,E1 -14127.623,E2 -14127.623} C_VEL
LIN {X 0,Y 339.194,Z 473.209,A -85,B 0,C 180,E1 -14128.811,E2 -14128.811} C_VEL
LIN {X 0,Y 339.3,Z 472.819,A -85,B 0,C 180,E1 -14129.999,E2 -14129.999} C_VEL
LIN {X 0,Y 339.294,Z 472.054,A -85,B 0,C 180,E1 -14131.186,E2 -14131.186} C_VEL
LIN {X 0,Y 339.128,Z 471.044,A -85,B 0,C 180,E1 -14133.563,E2 -14133.563} C_VEL
LIN {X 0,Y 339.114,Z 469.949,A -85,B 0,C 180,E1 -14134.754,E2 -14134.754} C_VEL
LIN {X 0,Y 339.169,Z 468.398,A -85,B 0,C 180,E1 -14135.946,E2 -14135.946} C_VEL
LIN {X 0,Y 339.338,Z 465.286,A -85,B 0,C 180,E1 -14137.735,E2 -14137.735} C_VEL
LIN {X 0,Y 339.718,Z 461.118,A -85,B 0,C 180,E1 -14139.525,E2 -14139.525} C_VEL
LIN {X 0,Y 340.453,Z 454.762,A -85,B 0,C 180,E1 -14141.61,E2 -14141.61} C_VEL
LIN {X 0,Y 341.572,Z 447.857,A -85,B 0,C 180,E1 -14143.382,E2 -14143.382} C_VEL
LIN {X 0,Y 342.726,Z 439.218,A -85,B 0,C 180,E1 -14145.155,E2 -14145.155} C_VEL
LIN {X 0,Y 344.034,Z 430.373,A -85,B 0,C 180,E1 -14146.617,E2 -14146.617} C_VEL
LIN {X 0,Y 345.562,Z 420.653,A -85,B 0,C 180,E1 -14147.914,E2 -14147.914} C_VEL
LIN {X 0,Y 346.989,Z 409.948,A -85,B 0,C 180,E1 -14149.061,E2 -14149.061} C_VEL
LIN {X 0,Y 348.334,Z 397.962,A -85,B 0,C 180,E1 -14150.058,E2 -14150.058} C_VEL
LIN {X 0,Y 349.617,Z 385.43,A -85,B 0,C 180,E1 -14150.826,E2 -14150.826} C_VEL
LIN {X 0,Y 350.604,Z 372.2,A -85,B 0,C 180,E1 -14151.369,E2 -14151.369} C_VEL
LIN {X 0,Y 351.072,Z 355.495,A -85,B 0,C 180,E1 -14151.78,E2 -14151.78} C_VEL
LIN {X 0,Y 352.176,Z 299.865,A -85,B 0,C 180,E1 -14152.951,E2 -14152.951} C_VEL
LIN {X 0,Y 349.492,Z 280.321,A -85,B 0,C 180,E1 -14153.622,E2 -14153.622} C_VEL
LIN {X 0,Y 343.988,Z 248.665,A -85,B 0,C 180,E1 -14154.88,E2 -14154.88} C_VEL
LIN {X 0,Y 344.26,Z 245.227,A -85,B 0,C 180,E1 -14155.693,E2 -14155.693} C_VEL
LIN {X 0,Y 342.468,Z 235.404,A -85,B 0,C 180,E1 -14158.162,E2 -14158.162} C_VEL
LIN {X 0,Y 340.752,Z 227.042,A -85,B 0,C 180,E1 -14160.365,E2 -14160.365} C_VEL
LIN {X 0,Y 340.718,Z 227.014,A -85,B 0,C 180,E1 -14164.403,E2 -14164.403} C_VEL
LIN {X 0,Y 340.713,Z 227.037,A -85,B 0,C 180,E1 -14168.228,E2 -14168.228} C_VEL
LIN {X 0,Y 340.687,Z 227.043,A -85,B 0,C 180,E1 -14172.043,E2 -14172.043} C_VEL
LIN {X 0,Y 340.645,Z 227.051,A -85,B 0,C 180,E1 -14176.226,E2 -14176.226} C_VEL
LIN {X 0,Y 340.663,Z 227.034,A -85,B 0,C 180,E1 -14178.687,E2 -14178.687} C_VEL
LIN {X 0,Y 340.711,Z 227.041,A -85,B 0,C 180,E1 -14181.77,E2 -14181.77} C_VEL
LIN {X 0,Y 340.715,Z 227.032,A -85,B 0,C 180,E1 -14185.595,E2 -14185.595} C_VEL
LIN {X 0,Y 340.686,Z 227.035,A -85,B 0,C 180,E1 -14188.954,E2 -14188.954} C_VEL
LIN {X 0,Y 340.703,Z 227.036,A -85,B 0,C 180,E1 -14193.011,E2 -14193.011} C_VEL
LIN {X 0,Y 340.73,Z 227.031,A -85,B 0,C 180,E1 -14195.637,E2 -14195.637} C_VEL
LIN {X 0,Y 340.719,Z 227.025,A -85,B 0,C 180,E1 -14199.473,E2 -14199.473} C_VEL
LIN {X 0,Y 340.783,Z 227.031,A -85,B 0,C 180,E1 -14201.98,E2 -14201.98} C_VEL
LIN {X 0,Y 340.844,Z 226.999,A -85,B 0,C 180,E1 -14205.716,E2 -14205.716} C_VEL
LIN {X 0,Y 340.838,Z 227.027,A -85,B 0,C 180,E1 -14209.305,E2 -14209.305} C_VEL
LIN {X 0,Y 340.988,Z 226.994,A -85,B 0,C 180,E1 -14212.897,E2 -14212.897} C_VEL
LIN {X 0,Y 340.809,Z 227.006,A -85,B 0,C 180,E1 -14215.269,E2 -14215.269} C_VEL
LIN {X 0,Y 341.146,Z 226.983,A -85,B 0,C 180,E1 -14217.639,E2 -14217.639} C_VEL
LIN {X 0,Y 341.103,Z 226.98,A -85,B 0,C 180,E1 -14221.181,E2 -14221.181} C_VEL
LIN {X 0,Y 341.12,Z 226.964,A -85,B 0,C 180,E1 -14222.362,E2 -14222.362} C_VEL
LIN {X 0,Y 341.05,Z 226.996,A -85,B 0,C 180,E1 -14227.103,E2 -14227.103} C_VEL
LIN {X 0,Y 340.862,Z 226.999,A -85,B 0,C 180,E1 -14230.694,E2 -14230.694} C_VEL
LIN {X 0,Y 340.855,Z 227.023,A -85,B 0,C 180,E1 -14234.326,E2 -14234.326} C_VEL
LIN {X 0,Y 340.778,Z 227.022,A -85,B 0,C 180,E1 -14238.441,E2 -14238.441} C_VEL
LIN {X 0,Y 340.747,Z 227.035,A -85,B 0,C 180,E1 -14241.858,E2 -14241.858} C_VEL
LIN {X 0,Y 340.766,Z 227.034,A -85,B 0,C 180,E1 -14245.665,E2 -14245.665} C_VEL
LIN {X 0,Y 340.722,Z 227.035,A -85,B 0,C 180,E1 -14248.322,E2 -14248.322} C_VEL
LIN {X 0,Y 340.692,Z 227.045,A -85,B 0,C 180,E1 -14251.046,E2 -14251.046} C_VEL
LIN {X 0,Y 340.713,Z 227.041,A -85,B 0,C 180,E1 -14255.28,E2 -14255.28} C_VEL
LIN {X 0,Y 340.706,Z 227.038,A -85,B 0,C 180,E1 -14258.387,E2 -14258.387} C_VEL
LIN {X 0,Y 340.695,Z 227.04,A -85,B 0,C 180,E1 -14262.047,E2 -14262.047} C_VEL
LIN {X 0,Y 340.649,Z 227.053,A -85,B 0,C 180,E1 -14266.228,E2 -14266.228} C_VEL
LIN {X 0,Y 340.686,Z 227.044,A -85,B 0,C 180,E1 -14269.754,E2 -14269.754} C_VEL
LIN {X 0,Y 340.727,Z 227.045,A -85,B 0,C 180,E1 -14270.736,E2 -14270.736} C_VEL
LIN {X 0,Y 341.821,Z 230.007,A -85,B 0,C 180,E1 -14270.922,E2 -14270.922} C_VEL
LIN {X 0,Y 349.737,Z 245.378,A -85,B 0,C 180,E1 -14272.01,E2 -14272.01} C_VEL
LIN {X 0,Y 353.365,Z 254.4,A -85,B 0,C 180,E1 -14272.532,E2 -14272.532} C_VEL
LIN {X 0,Y 353.805,Z 257.888,A -85,B 0,C 180,E1 -14272.649,E2 -14272.649} C_VEL
LIN {X 0,Y 351.747,Z 338.734,A -85,B 0,C 180,E1 -14274.328,E2 -14274.328} C_VEL
LIN {X 0,Y 351.144,Z 351.956,A -85,B 0,C 180,E1 -14274.818,E2 -14274.818} C_VEL
LIN {X 0,Y 350.367,Z 363.773,A -85,B 0,C 180,E1 -14275.483,E2 -14275.483} C_VEL
LIN {X 0,Y 349.157,Z 375.854,A -85,B 0,C 180,E1 -14276.392,E2 -14276.392} C_VEL
LIN {X 0,Y 347.951,Z 386.836,A -85,B 0,C 180,E1 -14277.469,E2 -14277.469} C_VEL
LIN {X 0,Y 346.547,Z 396.597,A -85,B 0,C 180,E1 -14278.657,E2 -14278.657} C_VEL
LIN {X 0,Y 345.162,Z 405.96,A -85,B 0,C 180,E1 -14280.077,E2 -14280.077} C_VEL
LIN {X 0,Y 343.884,Z 414.21,A -85,B 0,C 180,E1 -14281.617,E2 -14281.617} C_VEL
LIN {X 0,Y 342.503,Z 422.323,A -85,B 0,C 180,E1 -14283.495,E2 -14283.495} C_VEL
LIN {X 0,Y 341.502,Z 428.289,A -85,B 0,C 180,E1 -14285.248,E2 -14285.248} C_VEL
LIN {X 0,Y 340.731,Z 432.855,A -85,B 0,C 180,E1 -14286.929,E2 -14286.929} C_VEL
LIN {X 0,Y 340.221,Z 435.962,A -85,B 0,C 180,E1 -14288.37,E2 -14288.37} C_VEL
LIN {X 0,Y 339.878,Z 437.817,A -85,B 0,C 180,E1 -14289.421,E2 -14289.421} C_VEL
LIN {X 0,Y 339.531,Z 439.532,A -85,B 0,C 180,E1 -14290.661,E2 -14290.661} C_VEL
LIN {X 0,Y 339.264,Z 441.181,A -85,B 0,C 180,E1 -14292.349,E2 -14292.349} C_VEL
LIN {X 0,Y 339.038,Z 442.077,A -85,B 0,C 180,E1 -14294.368,E2 -14294.368} C_VEL
LIN {X 0,Y 338.982,Z 442.068,A -85,B 0,C 180,E1 -14295.595,E2 -14295.595} C_VEL
LIN {X 0,Y 339.03,Z 441.574,A -85,B 0,C 180,E1 -14296.984,E2 -14296.984} C_VEL
LIN {X 0,Y 339.103,Z 439.545,A -85,B 0,C 180,E1 -14299.251,E2 -14299.251} C_VEL
LIN {X 0,Y 339.346,Z 436.843,A -85,B 0,C 180,E1 -14301.066,E2 -14301.066} C_VEL
LIN {X 0,Y 339.733,Z 432.32,A -85,B 0,C 180,E1 -14303.206,E2 -14303.206} C_VEL
LIN {X 0,Y 340.027,Z 428.271,A -85,B 0,C 180,E1 -14304.665,E2 -14304.665} C_VEL
LIN {X 0,Y 340.641,Z 422.156,A -85,B 0,C 180,E1 -14306.453,E2 -14306.453} C_VEL
LIN {X 0,Y 341.376,Z 414.509,A -85,B 0,C 180,E1 -14308.232,E2 -14308.232} C_VEL
LIN {X 0,Y 342.356,Z 404.953,A -85,B 0,C 180,E1 -14310.001,E2 -14310.001} C_VEL
LIN {X 0,Y 343.36,Z 395.035,A -85,B 0,C 180,E1 -14311.467,E2 -14311.467} C_VEL
LIN {X 0,Y 344.506,Z 383.454,A -85,B 0,C 180,E1 -14312.822,E2 -14312.822} C_VEL
LIN {X 0,Y 345.352,Z 372.801,A -85,B 0,C 180,E1 -14313.809,E2 -14313.809} C_VEL
LIN {X 0,Y 346.039,Z 360.857,A -85,B 0,C 180,E1 -14314.661,E2 -14314.661} C_VEL
LIN {X 0,Y 346.615,Z 347.523,A -85,B 0,C 180,E1 -14315.346,E2 -14315.346} C_VEL
LIN {X 0,Y 347.032,Z 335.458,A -85,B 0,C 180,E1 -14315.74,E2 -14315.74} C_VEL
LIN {X 0,Y 348.436,Z 254.885,A -85,B 0,C 180,E1 -14317.394,E2 -14317.394} C_VEL
LIN {X 0,Y 345.949,Z 240.825,A -85,B 0,C 180,E1 -14317.828,E2 -14317.828} C_VEL
LIN {X 0,Y 341.004,Z 227.145,A -85,B 0,C 180,E1 -14318.398,E2 -14318.398} C_VEL
LIN {X 0,Y 340.855,Z 227.024,A -85,B 0,C 180,E1 -14321.9,E2 -14321.9} C_VEL
LIN {X 0,Y 340.826,Z 227.027,A -85,B 0,C 180,E1 -14325.551,E2 -14325.551} C_VEL
LIN {X 0,Y 340.844,Z 227.029,A -85,B 0,C 180,E1 -14328.467,E2 -14328.467} C_VEL
LIN {X 0,Y 340.723,Z 227.041,A -85,B 0,C 180,E1 -14331.664,E2 -14331.664} C_VEL
LIN {X 0,Y 340.081,Z 227.125,A -85,B 0,C 180,E1 -14332.652,E2 -14332.652} C_VEL
LIN {X 0,Y 337.199,Z 227.486,A -85,B 0,C 180,E1 -14334.257,E2 -14334.257} C_VEL
LIN {X 0,Y 334.745,Z 227.788,A -85,B 0,C 180,E1 -14335.557,E2 -14335.557} C_VEL
LIN {X 0,Y 333.704,Z 227.916,A -85,B 0,C 180,E1 -14336.564,E2 -14336.564} C_VEL
LIN {X 0,Y 333.627,Z 227.924,A -85,B 0,C 180,E1 -14336.905,E2 -14336.905} C_VEL
LIN {X 0,Y 333.663,Z 227.921,A -85,B 0,C 180,E1 -14340.367,E2 -14340.367} C_VEL
LIN {X 0,Y 333.643,Z 227.923,A -85,B 0,C 180,E1 -14343.209,E2 -14343.209} C_VEL
LIN {X 0,Y 333.679,Z 227.919,A -85,B 0,C 180,E1 -14346.14,E2 -14346.14} C_VEL
LIN {X 0,Y 333.607,Z 227.928,A -85,B 0,C 180,E1 -14349.199,E2 -14349.199} C_VEL
LIN {X 0,Y 333.632,Z 227.922,A -85,B 0,C 180,E1 -14352.499,E2 -14352.499} C_VEL
LIN {X 0,Y 333.599,Z 227.928,A -85,B 0,C 180,E1 -14355.955,E2 -14355.955} C_VEL
LIN {X 0,Y 333.608,Z 227.931,A -85,B 0,C 180,E1 -14359.325,E2 -14359.325} C_VEL
LIN {X 0,Y 333.666,Z 227.924,A -85,B 0,C 180,E1 -14363.17,E2 -14363.17} C_VEL
LIN {X 0,Y 333.678,Z 227.921,A -85,B 0,C 180,E1 -14365.341,E2 -14365.341} C_VEL
LIN {X 0,Y 333.626,Z 227.924,A -85,B 0,C 180,E1 -14368.221,E2 -14368.221} C_VEL
LIN {X 0,Y 333.654,Z 227.923,A -85,B 0,C 180,E1 -14371.022,E2 -14371.022} C_VEL
LIN {X 0,Y 333.669,Z 227.922,A -85,B 0,C 180,E1 -14375.086,E2 -14375.086} C_VEL
LIN {X 0,Y 333.743,Z 227.968,A -85,B 0,C 180,E1 -14376.085,E2 -14376.085} C_VEL
LIN {X 0,Y 334.438,Z 231.793,A -85,B 0,C 180,E1 -14377.235,E2 -14377.235} C_VEL
LIN {X 0,Y 338.5,Z 247.344,A -85,B 0,C 180,E1 -14377.871,E2 -14377.871} C_VEL
LIN {X 0,Y 340.167,Z 257.819,A -85,B 0,C 180,E1 -14378.255,E2 -14378.255} C_VEL
LIN {X 0,Y 337.623,Z 340.447,A -85,B 0,C 180,E1 -14380.703,E2 -14380.703} C_VEL
LIN {X 0,Y 337.175,Z 354.804,A -85,B 0,C 180,E1 -14381.387,E2 -14381.387} C_VEL
LIN {X 0,Y 336.613,Z 367.203,A -85,B 0,C 180,E1 -14382.22,E2 -14382.22} C_VEL
LIN {X 0,Y 335.827,Z 379.364,A -85,B 0,C 180,E1 -14383.276,E2 -14383.276} C_VEL
LIN {X 0,Y 335.11,Z 390.073,A -85,B 0,C 180,E1 -14384.441,E2 -14384.441} C_VEL
LIN {X 0,Y 334.427,Z 401.619,A -85,B 0,C 180,E1 -14386.014,E2 -14386.014} C_VEL
LIN {X 0,Y 333.744,Z 410.708,A -85,B 0,C 180,E1 -14387.535,E2 -14387.535} C_VEL
LIN {X 0,Y 333.125,Z 419.51,A -85,B 0,C 180,E1 -14389.362,E2 -14389.362} C_VEL
LIN {X 0,Y 332.688,Z 426.598,A -85,B 0,C 180,E1 -14391.19,E2 -14391.19} C_VEL
LIN {X 0,Y 332.432,Z 431.368,A -85,B 0,C 180,E1 -14392.712,E2 -14392.712} C_VEL
LIN {X 0,Y 332.229,Z 435.94,A -85,B 0,C 180,E1 -14394.537,E2 -14394.537} C_VEL
LIN {X 0,Y 332.16,Z 439.356,A -85,B 0,C 180,E1 -14396.36,E2 -14396.36} C_VEL
LIN {X 0,Y 332.086,Z 441.054,A -85,B 0,C 180,E1 -14397.574,E2 -14397.574} C_VEL
LIN {X 0,Y 332.092,Z 442.262,A -85,B 0,C 180,E1 -14398.787,E2 -14398.787} C_VEL
LIN {X 0,Y 332.173,Z 443.054,A -85,B 0,C 180,E1 -14400,E2 -14400} C_VEL
LIN {X 0,Y 332.313,Z 443.43,A -85,B 0,C 180,E1 -14401.212,E2 -14401.212} C_VEL
LIN {X 0,Y 332.493,Z 443.334,A -85,B 0,C 180,E1 -14402.423,E2 -14402.423} C_VEL
LIN {X 0,Y 332.76,Z 442.81,A -85,B 0,C 180,E1 -14403.632,E2 -14403.632} C_VEL
LIN {X 0,Y 333.074,Z 441.879,A -85,B 0,C 180,E1 -14404.841,E2 -14404.841} C_VEL
LIN {X 0,Y 333.352,Z 440.517,A -85,B 0,C 180,E1 -14406.051,E2 -14406.051} C_VEL
LIN {X 0,Y 333.47,Z 438.706,A -85,B 0,C 180,E1 -14407.264,E2 -14407.264} C_VEL
LIN {X 0,Y 334.67,Z 434.633,A -85,B 0,C 180,E1 -14409.246,E2 -14409.246} C_VEL
LIN {X 0,Y 335.552,Z 430.308,A -85,B 0,C 180,E1 -14410.865,E2 -14410.865} C_VEL
LIN {X 0,Y 336.89,Z 424.292,A -85,B 0,C 180,E1 -14412.653,E2 -14412.653} C_VEL
LIN {X 0,Y 338.443,Z 416.806,A -85,B 0,C 180,E1 -14414.429,E2 -14414.429} C_VEL
LIN {X 0,Y 340.239,Z 407.486,A -85,B 0,C 180,E1 -14416.192,E2 -14416.192} C_VEL
LIN {X 0,Y 342.205,Z 396.891,A -85,B 0,C 180,E1 -14417.788,E2 -14417.788} C_VEL
LIN {X 0,Y 344.213,Z 384.818,A -85,B 0,C 180,E1 -14419.222,E2 -14419.222} C_VEL
LIN {X 0,Y 345.682,Z 374.387,A -85,B 0,C 180,E1 -14420.22,E2 -14420.22} C_VEL
LIN {X 0,Y 347.334,Z 360.534,A -85,B 0,C 180,E1 -14421.244,E2 -14421.244} C_VEL
LIN {X 0,Y 348.516,Z 347.769,A -85,B 0,C 180,E1 -14421.943,E2 -14421.943} C_VEL
LIN {X 0,Y 349.842,Z 329.137,A -85,B 0,C 180,E1 -14422.633,E2 -14422.633} C_VEL
LIN {X 0,Y 354.658,Z 270.023,A -85,B 0,C 180,E1 -14424.65,E2 -14424.65} C_VEL
LIN {X 0,Y 349.849,Z 260.202,A -85,B 0,C 180,E1 -14425.926,E2 -14425.926} C_VEL
LIN {X 0,Y 345.609,Z 252.853,A -85,B 0,C 180,E1 -14427.108,E2 -14427.108} C_VEL
LIN {X 0,Y 342.815,Z 248.486,A -85,B 0,C 180,E1 -14427.931,E2 -14427.931} C_VEL
LIN {X 0,Y 340.438,Z 244.868,A -85,B 0,C 180,E1 -14428.672,E2 -14428.672} C_VEL
LIN {X 0,Y 337.875,Z 241.347,A -85,B 0,C 180,E1 -14429.505,E2 -14429.505} C_VEL
LIN {X 0,Y 337.5,Z 240.578,A -85,B 0,C 180,E1 -14429.671,E2 -14429.671} C_VEL
LIN {X 0,Y 336.433,Z 236.634,A -85,B 0,C 180,E1 -14432.897,E2 -14432.897} C_VEL
LIN {X 0,Y 335.632,Z 234.085,A -85,B 0,C 180,E1 -14435.895,E2 -14435.895} C_VEL
LIN {X 0,Y 335.115,Z 232.557,A -85,B 0,C 180,E1 -14438.988,E2 -14438.988} C_VEL
LIN {X 0,Y 334.995,Z 232.208,A -85,B 0,C 180,E1 -14442.171,E2 -14442.171} C_VEL
LIN {X 0,Y 335.36,Z 233.175,A -85,B 0,C 180,E1 -14445.441,E2 -14445.441} C_VEL
LIN {X 0,Y 335.871,Z 234.948,A -85,B 0,C 180,E1 -14447.963,E2 -14447.963} C_VEL
LIN {X 0,Y 337.046,Z 238.446,A -85,B 0,C 180,E1 -14451.276,E2 -14451.276} C_VEL
LIN {X 0,Y 337.802,Z 240.671,A -85,B 0,C 180,E1 -14452.889,E2 -14452.889} C_VEL
LIN {X 0,Y 339.247,Z 246.01,A -85,B 0,C 180,E1 -14455.988,E2 -14455.988} C_VEL
LIN {X 0,Y 340.759,Z 252.429,A -85,B 0,C 180,E1 -14458.96,E2 -14458.96} C_VEL
LIN {X 0,Y 341.495,Z 255.886,A -85,B 0,C 180,E1 -14460.289,E2 -14460.289} C_VEL
LIN {X 0,Y 343.842,Z 260.593,A -85,B 0,C 180,E1 -14461.043,E2 -14461.043} C_VEL
LIN {X 0,Y 346.581,Z 266.517,A -85,B 0,C 180,E1 -14461.885,E2 -14461.885} C_VEL
LIN {X 0,Y 349.182,Z 278.02,A -85,B 0,C 180,E1 -14462.934,E2 -14462.934} C_VEL
LIN {X 0,Y 351.644,Z 292.778,A -85,B 0,C 180,E1 -14464.044,E2 -14464.044} C_VEL
LIN {X 0,Y 352.64,Z 303.35,A -85,B 0,C 180,E1 -14464.681,E2 -14464.681} C_VEL
LIN {X 0,Y 347.623,Z 370.34,A -85,B 0,C 180,E1 -14466.977,E2 -14466.977} C_VEL
LIN {X 0,Y 345.986,Z 384.481,A -85,B 0,C 180,E1 -14467.69,E2 -14467.69} C_VEL
LIN {X 0,Y 344.205,Z 397.491,A -85,B 0,C 180,E1 -14468.593,E2 -14468.593} C_VEL
LIN {X 0,Y 342.232,Z 410.013,A -85,B 0,C 180,E1 -14469.723,E2 -14469.723} C_VEL
LIN {X 0,Y 340.128,Z 422.508,A -85,B 0,C 180,E1 -14471.163,E2 -14471.163} C_VEL
LIN {X 0,Y 338.443,Z 431.701,A -85,B 0,C 180,E1 -14472.475,E2 -14472.475} C_VEL
LIN {X 0,Y 336.486,Z 441.823,A -85,B 0,C 180,E1 -14474.244,E2 -14474.244} C_VEL
LIN {X 0,Y 335.114,Z 450.044,A -85,B 0,C 180,E1 -14476.043,E2 -14476.043} C_VEL
LIN {X 0,Y 333.802,Z 456.72,A -85,B 0,C 180,E1 -14477.844,E2 -14477.844} C_VEL
LIN {X 0,Y 333.01,Z 462.076,A -85,B 0,C 180,E1 -14479.665,E2 -14479.665} C_VEL
LIN {X 0,Y 332.461,Z 466.282,A -85,B 0,C 180,E1 -14481.489,E2 -14481.489} C_VEL
LIN {X 0,Y 332.186,Z 468.482,A -85,B 0,C 180,E1 -14482.706,E2 -14482.706} C_VEL
LIN {X 0,Y 332.034,Z 470.527,A -85,B 0,C 180,E1 -14484.169,E2 -14484.169} C_VEL
LIN {X 0,Y 332.009,Z 472.378,A -85,B 0,C 180,E1 -14486.358,E2 -14486.358} C_VEL
LIN {X 0,Y 331.98,Z 472.807,A -85,B 0,C 180,E1 -14487.572,E2 -14487.572} C_VEL
LIN {X 0,Y 332.1,Z 472.801,A -85,B 0,C 180,E1 -14488.786,E2 -14488.786} C_VEL
LIN {X 0,Y 332.194,Z 471.746,A -85,B 0,C 180,E1 -14491.211,E2 -14491.211} C_VEL
LIN {X 0,Y 332.049,Z 470.78,A -85,B 0,C 180,E1 -14493.639,E2 -14493.639} C_VEL
LIN {X 0,Y 332.071,Z 468.462,A -85,B 0,C 180,E1 -14495.893,E2 -14495.893} C_VEL
LIN {X 0,Y 332.263,Z 465.136,A -85,B 0,C 180,E1 -14497.901,E2 -14497.901} C_VEL
LIN {X 0,Y 332.699,Z 461.022,A -85,B 0,C 180,E1 -14499.728,E2 -14499.728} C_VEL
LIN {X 0,Y 333.48,Z 454.726,A -85,B 0,C 180,E1 -14501.856,E2 -14501.856} C_VEL
LIN {X 0,Y 334.636,Z 447.887,A -85,B 0,C 180,E1 -14503.665,E2 -14503.665} C_VEL
LIN {X 0,Y 335.785,Z 439.862,A -85,B 0,C 180,E1 -14505.378,E2 -14505.378} C_VEL
LIN {X 0,Y 337.25,Z 430.599,A -85,B 0,C 180,E1 -14506.961,E2 -14506.961} C_VEL
LIN {X 0,Y 338.965,Z 419.827,A -85,B 0,C 180,E1 -14508.431,E2 -14508.431} C_VEL
LIN {X 0,Y 340.529,Z 408.951,A -85,B 0,C 180,E1 -14509.594,E2 -14509.594} C_VEL
LIN {X 0,Y 341.92,Z 396.803,A -85,B 0,C 180,E1 -14510.608,E2 -14510.608} C_VEL
LIN {X 0,Y 343.15,Z 385.304,A -85,B 0,C 180,E1 -14511.316,E2 -14511.316} C_VEL
LIN {X 0,Y 344.131,Z 373.024,A -85,B 0,C 180,E1 -14511.842,E2 -14511.842} C_VEL
LIN {X 0,Y 344.623,Z 357.805,A -85,B 0,C 180,E1 -14512.241,E2 -14512.241} C_VEL
LIN {X 0,Y 345.837,Z 300.634,A -85,B 0,C 180,E1 -14513.466,E2 -14513.466} C_VEL
LIN {X 0,Y 342.824,Z 278.731,A -85,B 0,C 180,E1 -14514.244,E2 -14514.244} C_VEL
LIN {X 0,Y 337.228,Z 247.058,A -85,B 0,C 180,E1 -14515.551,E2 -14515.551} C_VEL
LIN {X 0,Y 336.381,Z 241.098,A -85,B 0,C 180,E1 -14517.062,E2 -14517.062} C_VEL
LIN {X 0,Y 333.702,Z 227.919,A -85,B 0,C 180,E1 -14520.535,E2 -14520.535} C_VEL
LIN {X 0,Y 333.681,Z 227.895,A -85,B 0,C 180,E1 -14524.773,E2 -14524.773} C_VEL
LIN {X 0,Y 333.638,Z 227.924,A -85,B 0,C 180,E1 -14527.651,E2 -14527.651} C_VEL
LIN {X 0,Y 333.598,Z 227.93,A -85,B 0,C 180,E1 -14530.773,E2 -14530.773} C_VEL
LIN {X 0,Y 333.586,Z 227.926,A -85,B 0,C 180,E1 -14534.249,E2 -14534.249} C_VEL
LIN {X 0,Y 333.631,Z 227.913,A -85,B 0,C 180,E1 -14537.617,E2 -14537.617} C_VEL
LIN {X 0,Y 333.627,Z 227.928,A -85,B 0,C 180,E1 -14541.205,E2 -14541.205} C_VEL
LIN {X 0,Y 333.667,Z 227.899,A -85,B 0,C 180,E1 -14543.86,E2 -14543.86} C_VEL
LIN {X 0,Y 333.636,Z 227.923,A -85,B 0,C 180,E1 -14547.412,E2 -14547.412} C_VEL
LIN {X 0,Y 333.624,Z 227.901,A -85,B 0,C 180,E1 -14551.02,E2 -14551.02} C_VEL
LIN {X 0,Y 333.686,Z 227.912,A -85,B 0,C 180,E1 -14555.088,E2 -14555.088} C_VEL
LIN {X 0,Y 333.653,Z 227.897,A -85,B 0,C 180,E1 -14559.018,E2 -14559.018} C_VEL
LIN {X 0,Y 333.732,Z 227.91,A -85,B 0,C 180,E1 -14561.586,E2 -14561.586} C_VEL
LIN {X 0,Y 333.799,Z 227.876,A -85,B 0,C 180,E1 -14565.577,E2 -14565.577} C_VEL
LIN {X 0,Y 333.808,Z 227.903,A -85,B 0,C 180,E1 -14569.077,E2 -14569.077} C_VEL
LIN {X 0,Y 333.944,Z 227.872,A -85,B 0,C 180,E1 -14572.746,E2 -14572.746} C_VEL
LIN {X 0,Y 333.775,Z 227.881,A -85,B 0,C 180,E1 -14575.169,E2 -14575.169} C_VEL
LIN {X 0,Y 334.083,Z 227.863,A -85,B 0,C 180,E1 -14577.589,E2 -14577.589} C_VEL
LIN {X 0,Y 334.071,Z 227.855,A -85,B 0,C 180,E1 -14581.206,E2 -14581.206} C_VEL
LIN {X 0,Y 333.804,Z 227.877,A -85,B 0,C 180,E1 -14583.622,E2 -14583.622} C_VEL
LIN {X 0,Y 333.982,Z 227.874,A -85,B 0,C 180,E1 -14586.65,E2 -14586.65} C_VEL
LIN {X 0,Y 333.842,Z 227.875,A -85,B 0,C 180,E1 -14589.696,E2 -14589.696} C_VEL
LIN {X 0,Y 333.789,Z 227.901,A -85,B 0,C 180,E1 -14593.392,E2 -14593.392} C_VEL
LIN {X 0,Y 333.711,Z 227.895,A -85,B 0,C 180,E1 -14597.148,E2 -14597.148} C_VEL
LIN {X 0,Y 333.713,Z 227.911,A -85,B 0,C 180,E1 -14599.692,E2 -14599.692} C_VEL
LIN {X 0,Y 333.686,Z 227.911,A -85,B 0,C 180,E1 -14602.279,E2 -14602.279} C_VEL
LIN {X 0,Y 333.728,Z 227.914,A -85,B 0,C 180,E1 -14606.247,E2 -14606.247} C_VEL
LIN {X 0,Y 333.684,Z 227.908,A -85,B 0,C 180,E1 -14608.975,E2 -14608.975} C_VEL
LIN {X 0,Y 333.638,Z 227.926,A -85,B 0,C 180,E1 -14612.588,E2 -14612.588} C_VEL
LIN {X 0,Y 333.671,Z 227.924,A -85,B 0,C 180,E1 -14616.14,E2 -14616.14} C_VEL
LIN {X 0,Y 333.642,Z 227.922,A -85,B 0,C 180,E1 -14619.194,E2 -14619.194} C_VEL
LIN {X 0,Y 333.629,Z 227.922,A -85,B 0,C 180,E1 -14622.501,E2 -14622.501} C_VEL
LIN {X 0,Y 333.594,Z 227.931,A -85,B 0,C 180,E1 -14625.957,E2 -14625.957} C_VEL
LIN {X 0,Y 333.644,Z 227.922,A -85,B 0,C 180,E1 -14629.317,E2 -14629.317} C_VEL
LIN {X 0,Y 333.666,Z 227.963,A -85,B 0,C 180,E1 -14630.07,E2 -14630.07} C_VEL
LIN {X 0,Y 334.598,Z 230.675,A -85,B 0,C 180,E1 -14630.232,E2 -14630.232} C_VEL
LIN {X 0,Y 336.283,Z 233.637,A -85,B 0,C 180,E1 -14630.472,E2 -14630.472} C_VEL
LIN {X 0,Y 344.417,Z 249.472,A -85,B 0,C 180,E1 -14631.626,E2 -14631.626} C_VEL
LIN {X 0,Y 347.317,Z 256.717,A -85,B 0,C 180,E1 -14632.057,E2 -14632.057} C_VEL
LIN {X 0,Y 347.404,Z 263.896,A -85,B 0,C 180,E1 -14632.231,E2 -14632.231} C_VEL
LIN {X 0,Y 345.396,Z 338.499,A -85,B 0,C 180,E1 -14633.803,E2 -14633.803} C_VEL
LIN {X 0,Y 344.785,Z 351.857,A -85,B 0,C 180,E1 -14634.3,E2 -14634.3} C_VEL
LIN {X 0,Y 344.068,Z 362.256,A -85,B 0,C 180,E1 -14634.874,E2 -14634.874} C_VEL
LIN {X 0,Y 342.969,Z 373.674,A -85,B 0,C 180,E1 -14635.702,E2 -14635.702} C_VEL
LIN {X 0,Y 341.638,Z 385.105,A -85,B 0,C 180,E1 -14636.791,E2 -14636.791} C_VEL
LIN {X 0,Y 340.016,Z 396.402,A -85,B 0,C 180,E1 -14638.153,E2 -14638.153} C_VEL
LIN {X 0,Y 338.672,Z 404.978,A -85,B 0,C 180,E1 -14639.443,E2 -14639.443} C_VEL
LIN {X 0,Y 337.223,Z 413.801,A -85,B 0,C 180,E1 -14641.083,E2 -14641.083} C_VEL
LIN {X 0,Y 335.824,Z 421.772,A -85,B 0,C 180,E1 -14642.925,E2 -14642.925} C_VEL
LIN {X 0,Y 334.827,Z 427.259,A -85,B 0,C 180,E1 -14644.499,E2 -14644.499} C_VEL
LIN {X 0,Y 333.859,Z 432.644,A -85,B 0,C 180,E1 -14646.426,E2 -14646.426} C_VEL
LIN {X 0,Y 333.212,Z 436.299,A -85,B 0,C 180,E1 -14648.132,E2 -14648.132} C_VEL
LIN {X 0,Y 332.575,Z 439.593,A -85,B 0,C 180,E1 -14650.24,E2 -14650.24} C_VEL
LIN {X 0,Y 332.22,Z 441.487,A -85,B 0,C 180,E1 -14652.17,E2 -14652.17} C_VEL
LIN {X 0,Y 331.97,Z 442.369,A -85,B 0,C 180,E1 -14654.026,E2 -14654.026} C_VEL
LIN {X 0,Y 331.893,Z 442.417,A -85,B 0,C 180,E1 -14655.281,E2 -14655.281} C_VEL
LIN {X 0,Y 331.941,Z 441.907,A -85,B 0,C 180,E1 -14656.892,E2 -14656.892} C_VEL
LIN {X 0,Y 332.012,Z 440.117,A -85,B 0,C 180,E1 -14659.019,E2 -14659.019} C_VEL
LIN {X 0,Y 332.205,Z 437.534,A -85,B 0,C 180,E1 -14660.872,E2 -14660.872} C_VEL
LIN {X 0,Y 332.66,Z 432.807,A -85,B 0,C 180,E1 -14663.2,E2 -14663.2} C_VEL
LIN {X 0,Y 333.066,Z 427.389,A -85,B 0,C 180,E1 -14665.16,E2 -14665.16} C_VEL
LIN {X 0,Y 333.754,Z 420.933,A -85,B 0,C 180,E1 -14666.984,E2 -14666.984} C_VEL
LIN {X 0,Y 334.574,Z 412.925,A -85,B 0,C 180,E1 -14668.798,E2 -14668.798} C_VEL
LIN {X 0,Y 335.451,Z 404.735,A -85,B 0,C 180,E1 -14670.301,E2 -14670.301} C_VEL
LIN {X 0,Y 336.519,Z 394.649,A -85,B 0,C 180,E1 -14671.796,E2 -14671.796} C_VEL
LIN {X 0,Y 337.638,Z 383.343,A -85,B 0,C 180,E1 -14673.133,E2 -14673.133} C_VEL
LIN {X 0,Y 338.573,Z 371.806,A -85,B 0,C 180,E1 -14674.199,E2 -14674.199} C_VEL
LIN {X 0,Y 339.261,Z 359.697,A -85,B 0,C 180,E1 -14675.052,E2 -14675.052} C_VEL
LIN {X 0,Y 339.874,Z 346.57,A -85,B 0,C 180,E1 -14675.712,E2 -14675.712} C_VEL
LIN {X 0,Y 340.262,Z 332.859,A -85,B 0,C 180,E1 -14676.129,E2 -14676.129} C_VEL
LIN {X 0,Y 341.731,Z 256.099,A -85,B 0,C 180,E1 -14677.724,E2 -14677.724} C_VEL
LIN {X 0,Y 339.38,Z 242.713,A -85,B 0,C 180,E1 -14678.147,E2 -14678.147} C_VEL
LIN {X 0,Y 333.894,Z 227.895,A -85,B 0,C 180,E1 -14678.81,E2 -14678.81} C_VEL
LIN {X 0,Y 333.797,Z 227.905,A -85,B 0,C 180,E1 -14682.156,E2 -14682.156} C_VEL
LIN {X 0,Y 333.784,Z 227.906,A -85,B 0,C 180,E1 -14685.887,E2 -14685.887} C_VEL
LIN {X 0,Y 333.803,Z 227.905,A -85,B 0,C 180,E1 -14688.656,E2 -14688.656} C_VEL
LIN {X 0,Y 333.657,Z 227.925,A -85,B 0,C 180,E1 -14692.282,E2 -14692.282} C_VEL
LIN {X 0,Y 333.665,Z 227.919,A -85,B 0,C 180,E1 -14695.079,E2 -14695.079} C_VEL
LIN {X 0,Y 333.627,Z 227.924,A -85,B 0,C 180,E1 -14696.905,E2 -14696.905} C_VEL
LIN {X 0,Y 332.969,Z 228.011,A -85,B 0,C 180,E1 -14697.914,E2 -14697.914} C_VEL
LIN {X 0,Y 330.085,Z 228.367,A -85,B 0,C 180,E1 -14699.553,E2 -14699.553} C_VEL
LIN {X 0,Y 327.657,Z 228.667,A -85,B 0,C 180,E1 -14700.882,E2 -14700.882} C_VEL
LIN {X 0,Y 326.652,Z 228.798,A -85,B 0,C 180,E1 -14701.91,E2 -14701.91} C_VEL
LIN {X 0,Y 326.591,Z 228.799,A -85,B 0,C 180,E1 -14702.259,E2 -14702.259} C_VEL
LIN {X 0,Y 326.617,Z 228.8,A -85,B 0,C 180,E1 -14705.521,E2 -14705.521} C_VEL
LIN {X 0,Y 326.577,Z 228.804,A -85,B 0,C 180,E1 -14709.219,E2 -14709.219} C_VEL
LIN {X 0,Y 326.578,Z 228.802,A -85,B 0,C 180,E1 -14712.971,E2 -14712.971} C_VEL
LIN {X 0,Y 326.578,Z 228.805,A -85,B 0,C 180,E1 -14717.03,E2 -14717.03} C_VEL
LIN {X 0,Y 326.587,Z 228.803,A -85,B 0,C 180,E1 -14721.386,E2 -14721.386} C_VEL
LIN {X 0,Y 326.623,Z 228.799,A -85,B 0,C 180,E1 -14724.852,E2 -14724.852} C_VEL
LIN {X 0,Y 326.608,Z 228.8,A -85,B 0,C 180,E1 -14727.455,E2 -14727.455} C_VEL
LIN {X 0,Y 326.593,Z 228.8,A -85,B 0,C 180,E1 -14730.334,E2 -14730.334} C_VEL
LIN {X 0,Y 326.601,Z 228.799,A -85,B 0,C 180,E1 -14733.134,E2 -14733.134} C_VEL
LIN {X 0,Y 326.67,Z 228.856,A -85,B 0,C 180,E1 -14735.957,E2 -14735.957} C_VEL
LIN {X 0,Y 327.276,Z 232.105,A -85,B 0,C 180,E1 -14736.945,E2 -14736.945} C_VEL
LIN {X 0,Y 331.778,Z 249.409,A -85,B 0,C 180,E1 -14737.676,E2 -14737.676} C_VEL
LIN {X 0,Y 333.225,Z 258.036,A -85,B 0,C 180,E1 -14738.003,E2 -14738.003} C_VEL
LIN {X 0,Y 330.608,Z 340.477,A -85,B 0,C 180,E1 -14740.519,E2 -14740.519} C_VEL
LIN {X 0,Y 330.159,Z 354.847,A -85,B 0,C 180,E1 -14741.218,E2 -14741.218} C_VEL
LIN {X 0,Y 329.62,Z 366.314,A -85,B 0,C 180,E1 -14741.991,E2 -14741.991} C_VEL
LIN {X 0,Y 328.832,Z 378.675,A -85,B 0,C 180,E1 -14743.07,E2 -14743.07} C_VEL
LIN {X 0,Y 328.005,Z 390.776,A -85,B 0,C 180,E1 -14744.408,E2 -14744.408} C_VEL
LIN {X 0,Y 327.295,Z 402.294,A -85,B 0,C 180,E1 -14746.02,E2 -14746.02} C_VEL
LIN {X 0,Y 326.634,Z 411.32,A -85,B 0,C 180,E1 -14747.574,E2 -14747.574} C_VEL
LIN {X 0,Y 326,Z 420.08,A -85,B 0,C 180,E1 -14749.441,E2 -14749.441} C_VEL
LIN {X 0,Y 325.561,Z 427.147,A -85,B 0,C 180,E1 -14751.308,E2 -14751.308} C_VEL
LIN {X 0,Y 325.283,Z 432.747,A -85,B 0,C 180,E1 -14753.175,E2 -14753.175} C_VEL
LIN {X 0,Y 325.138,Z 437.075,A -85,B 0,C 180,E1 -14755.04,E2 -14755.04} C_VEL
LIN {X 0,Y 325.088,Z 439.31,A -85,B 0,C 180,E1 -14756.281,E2 -14756.281} C_VEL
LIN {X 0,Y 324.999,Z 441.105,A -85,B 0,C 180,E1 -14757.521,E2 -14757.521} C_VEL
LIN {X 0,Y 324.994,Z 442.442,A -85,B 0,C 180,E1 -14758.761,E2 -14758.761} C_VEL
LIN {X 0,Y 325.077,Z 443.307,A -85,B 0,C 180,E1 -14760,E2 -14760} C_VEL
LIN {X 0,Y 325.223,Z 443.76,A -85,B 0,C 180,E1 -14761.238,E2 -14761.238} C_VEL
LIN {X 0,Y 325.426,Z 443.796,A -85,B 0,C 180,E1 -14762.475,E2 -14762.475} C_VEL
LIN {X 0,Y 325.722,Z 443.357,A -85,B 0,C 180,E1 -14763.711,E2 -14763.711} C_VEL
LIN {X 0,Y 326.051,Z 442.502,A -85,B 0,C 180,E1 -14764.946,E2 -14764.946} C_VEL
LIN {X 0,Y 326.339,Z 441.247,A -85,B 0,C 180,E1 -14766.181,E2 -14766.181} C_VEL
LIN {X 0,Y 326.481,Z 439.569,A -85,B 0,C 180,E1 -14767.421,E2 -14767.421} C_VEL
LIN {X 0,Y 327.736,Z 435.661,A -85,B 0,C 180,E1 -14769.444,E2 -14769.444} C_VEL
LIN {X 0,Y 329.163,Z 429.727,A -85,B 0,C 180,E1 -14771.703,E2 -14771.703} C_VEL
LIN {X 0,Y 330.635,Z 423.477,A -85,B 0,C 180,E1 -14773.522,E2 -14773.522} C_VEL
LIN {X 0,Y 332.362,Z 415.673,A -85,B 0,C 180,E1 -14775.326,E2 -14775.326} C_VEL
LIN {X 0,Y 334.374,Z 406.067,A -85,B 0,C 180,E1 -14777.113,E2 -14777.113} C_VEL
LIN {X 0,Y 336.579,Z 394.996,A -85,B 0,C 180,E1 -14778.726,E2 -14778.726} C_VEL
LIN {X 0,Y 338.495,Z 383.82,A -85,B 0,C 180,E1 -14780.034,E2 -14780.034} C_VEL
LIN {X 0,Y 340.206,Z 372.117,A -85,B 0,C 180,E1 -14781.126,E2 -14781.126} C_VEL
LIN {X 0,Y 341.829,Z 359.134,A -85,B 0,C 180,E1 -14782.061,E2 -14782.061} C_VEL
LIN {X 0,Y 343.031,Z 346.919,A -85,B 0,C 180,E1 -14782.715,E2 -14782.715} C_VEL
LIN {X 0,Y 344.648,Z 325.831,A -85,B 0,C 180,E1 -14783.498,E2 -14783.498} C_VEL
LIN {X 0,Y 349.294,Z 272.687,A -85,B 0,C 180,E1 -14785.376,E2 -14785.376} C_VEL
LIN {X 0,Y 344.444,Z 262.775,A -85,B 0,C 180,E1 -14786.77,E2 -14786.77} C_VEL
LIN {X 0,Y 339.972,Z 255.084,A -85,B 0,C 180,E1 -14788.129,E2 -14788.129} C_VEL
LIN {X 0,Y 336.665,Z 250.221,A -85,B 0,C 180,E1 -14789.197,E2 -14789.197} C_VEL
LIN {X 0,Y 333.814,Z 246.143,A -85,B 0,C 180,E1 -14790.203,E2 -14790.203} C_VEL
LIN {X 0,Y 331.058,Z 242.556,A -85,B 0,C 180,E1 -14791.241,E2 -14791.241} C_VEL
LIN {X 0,Y 330.629,Z 241.573,A -85,B 0,C 180,E1 -14791.521,E2 -14791.521} C_VEL
LIN {X 0,Y 329.942,Z 239.232,A -85,B 0,C 180,E1 -14793.824,E2 -14793.824} C_VEL
LIN {X 0,Y 329.31,Z 237.133,A -85,B 0,C 180,E1 -14796.696,E2 -14796.696} C_VEL
LIN {X 0,Y 328.93,Z 235.976,A -85,B 0,C 180,E1 -14799.865,E2 -14799.865} C_VEL
LIN {X 0,Y 328.942,Z 236.046,A -85,B 0,C 180,E1 -14803.133,E2 -14803.133} C_VEL
LIN {X 0,Y 329.237,Z 236.723,A -85,B 0,C 180,E1 -14805.215,E2 -14805.215} C_VEL
LIN {X 0,Y 329.852,Z 238.786,A -85,B 0,C 180,E1 -14808.222,E2 -14808.222} C_VEL
LIN {X 0,Y 330.533,Z 240.921,A -85,B 0,C 180,E1 -14810.365,E2 -14810.365} C_VEL
LIN {X 0,Y 331.592,Z 244.085,A -85,B 0,C 180,E1 -14812.839,E2 -14812.839} C_VEL
LIN {X 0,Y 332.936,Z 249.131,A -85,B 0,C 180,E1 -14815.85,E2 -14815.85} C_VEL
LIN {X 0,Y 334.268,Z 254.872,A -85,B 0,C 180,E1 -14818.574,E2 -14818.574} C_VEL
LIN {X 0,Y 336.871,Z 259.902,A -85,B 0,C 180,E1 -14819.53,E2 -14819.53} C_VEL
LIN {X 0,Y 338.442,Z 263.019,A -85,B 0,C 180,E1 -14820.074,E2 -14820.074} C_VEL
LIN {X 0,Y 340.679,Z 267.439,A -85,B 0,C 180,E1 -14820.808,E2 -14820.808} C_VEL
LIN {X 0,Y 342.299,Z 271.43,A -85,B 0,C 180,E1 -14821.356,E2 -14821.356} C_VEL
LIN {X 0,Y 344.983,Z 285.014,A -85,B 0,C 180,E1 -14822.588,E2 -14822.588} C_VEL
LIN {X 0,Y 346.837,Z 298.764,A -85,B 0,C 180,E1 -14823.597,E2 -14823.597} C_VEL
LIN {X 0,Y 347.191,Z 305.577,A -85,B 0,C 180,E1 -14823.983,E2 -14823.983} C_VEL
LIN {X 0,Y 341.997,Z 369.815,A -85,B 0,C 180,E1 -14826.255,E2 -14826.255} C_VEL
LIN {X 0,Y 340.241,Z 383.859,A -85,B 0,C 180,E1 -14826.971,E2 -14826.971} C_VEL
LIN {X 0,Y 338.379,Z 396.771,A -85,B 0,C 180,E1 -14827.885,E2 -14827.885} C_VEL
LIN {X 0,Y 336.225,Z 409.309,A -85,B 0,C 180,E1 -14829.024,E2 -14829.024} C_VEL
LIN {X 0,Y 333.957,Z 421.796,A -85,B 0,C 180,E1 -14830.482,E2 -14830.482} C_VEL
LIN {X 0,Y 331.761,Z 432.825,A -85,B 0,C 180,E1 -14832.11,E2 -14832.11} C_VEL
LIN {X 0,Y 329.716,Z 442.66,A -85,B 0,C 180,E1 -14833.912,E2 -14833.912} C_VEL
LIN {X 0,Y 328.254,Z 450.585,A -85,B 0,C 180,E1 -14835.745,E2 -14835.745} C_VEL
LIN {X 0,Y 326.861,Z 457.079,A -85,B 0,C 180,E1 -14837.582,E2 -14837.582} C_VEL
LIN {X 0,Y 326.011,Z 462.278,A -85,B 0,C 180,E1 -14839.44,E2 -14839.44} C_VEL
LIN {X 0,Y 325.426,Z 466.333,A -85,B 0,C 180,E1 -14841.304,E2 -14841.304} C_VEL
LIN {X 0,Y 325.14,Z 468.463,A -85,B 0,C 180,E1 -14842.547,E2 -14842.547} C_VEL
LIN {X 0,Y 324.946,Z 470.56,A -85,B 0,C 180,E1 -14844.21,E2 -14844.21} C_VEL
LIN {X 0,Y 324.934,Z 472.106,A -85,B 0,C 180,E1 -14846.278,E2 -14846.278} C_VEL
LIN {X 0,Y 324.895,Z 472.463,A -85,B 0,C 180,E1 -14847.519,E2 -14847.519} C_VEL
LIN {X 0,Y 325.009,Z 472.344,A -85,B 0,C 180,E1 -14848.76,E2 -14848.76} C_VEL
LIN {X 0,Y 325.18,Z 471.799,A -85,B 0,C 180,E1 -14849.999,E2 -14849.999} C_VEL
LIN {X 0,Y 324.983,Z 471.174,A -85,B 0,C 180,E1 -14852.478,E2 -14852.478} C_VEL
LIN {X 0,Y 324.971,Z 470.521,A -85,B 0,C 180,E1 -14853.719,E2 -14853.719} C_VEL
LIN {X 0,Y 324.995,Z 468.43,A -85,B 0,C 180,E1 -14855.874,E2 -14855.874} C_VEL
LIN {X 0,Y 325.203,Z 464.99,A -85,B 0,C 180,E1 -14858.074,E2 -14858.074} C_VEL
LIN {X 0,Y 325.67,Z 460.928,A -85,B 0,C 180,E1 -14859.94,E2 -14859.94} C_VEL
LIN {X 0,Y 326.518,Z 454.689,A -85,B 0,C 180,E1 -14862.113,E2 -14862.113} C_VEL
LIN {X 0,Y 327.726,Z 447.912,A -85,B 0,C 180,E1 -14863.959,E2 -14863.959} C_VEL
LIN {X 0,Y 328.868,Z 440.382,A -85,B 0,C 180,E1 -14865.63,E2 -14865.63} C_VEL
LIN {X 0,Y 330.489,Z 430.84,A -85,B 0,C 180,E1 -14867.319,E2 -14867.319} C_VEL
LIN {X 0,Y 332.255,Z 420.195,A -85,B 0,C 180,E1 -14868.817,E2 -14868.817} C_VEL
LIN {X 0,Y 333.872,Z 409.56,A -85,B 0,C 180,E1 -14870.001,E2 -14870.001} C_VEL
LIN {X 0,Y 335.341,Z 397.653,A -85,B 0,C 180,E1 -14871.031,E2 -14871.031} C_VEL
LIN {X 0,Y 336.731,Z 385.242,A -85,B 0,C 180,E1 -14871.823,E2 -14871.823} C_VEL
LIN {X 0,Y 337.817,Z 372.046,A -85,B 0,C 180,E1 -14872.393,E2 -14872.393} C_VEL
LIN {X 0,Y 338.371,Z 354.699,A -85,B 0,C 180,E1 -14872.837,E2 -14872.837} C_VEL
LIN {X 0,Y 339.57,Z 301.641,A -85,B 0,C 180,E1 -14873.992,E2 -14873.992} C_VEL
LIN {X 0,Y 336.568,Z 279.818,A -85,B 0,C 180,E1 -14874.791,E2 -14874.791} C_VEL
LIN {X 0,Y 331.097,Z 249.385,A -85,B 0,C 180,E1 -14876.072,E2 -14876.072} C_VEL
LIN {X 0,Y 329.949,Z 245.159,A -85,B 0,C 180,E1 -14876.346,E2 -14876.346} C_VEL
LIN {X 0,Y 327.212,Z 231.726,A -85,B 0,C 180,E1 -14879.916,E2 -14879.916} C_VEL
LIN {X 0,Y 326.68,Z 228.793,A -85,B 0,C 180,E1 -14880.719,E2 -14880.719} C_VEL
LIN {X 0,Y 326.602,Z 228.768,A -85,B 0,C 180,E1 -14884.018,E2 -14884.018} C_VEL
LIN {X 0,Y 326.618,Z 228.801,A -85,B 0,C 180,E1 -14887.236,E2 -14887.236} C_VEL
LIN {X 0,Y 326.539,Z 228.81,A -85,B 0,C 180,E1 -14891.123,E2 -14891.123} C_VEL
LIN {X 0,Y 326.554,Z 228.796,A -85,B 0,C 180,E1 -14893.525,E2 -14893.525} C_VEL
LIN {X 0,Y 326.567,Z 228.8,A -85,B 0,C 180,E1 -14897.028,E2 -14897.028} C_VEL
LIN {X 0,Y 326.575,Z 228.805,A -85,B 0,C 180,E1 -14901.385,E2 -14901.385} C_VEL
LIN {X 0,Y 326.611,Z 228.78,A -85,B 0,C 180,E1 -14904.851,E2 -14904.851} C_VEL
LIN {X 0,Y 326.6,Z 228.799,A -85,B 0,C 180,E1 -14907.455,E2 -14907.455} C_VEL
LIN {X 0,Y 326.573,Z 228.779,A -85,B 0,C 180,E1 -14910.332,E2 -14910.332} C_VEL
LIN {X 0,Y 326.624,Z 228.794,A -85,B 0,C 180,E1 -14914.511,E2 -14914.511} C_VEL
LIN {X 0,Y 326.605,Z 228.77,A -85,B 0,C 180,E1 -14918.543,E2 -14918.543} C_VEL
LIN {X 0,Y 326.654,Z 228.794,A -85,B 0,C 180,E1 -14922.47,E2 -14922.47} C_VEL
LIN {X 0,Y 326.747,Z 228.753,A -85,B 0,C 180,E1 -14926.314,E2 -14926.314} C_VEL
LIN {X 0,Y 326.774,Z 228.78,A -85,B 0,C 180,E1 -14930.093,E2 -14930.093} C_VEL
LIN {X 0,Y 326.93,Z 228.734,A -85,B 0,C 180,E1 -14933.83,E2 -14933.83} C_VEL
LIN {X 0,Y 327.023,Z 228.742,A -85,B 0,C 180,E1 -14937.537,E2 -14937.537} C_VEL
LIN {X 0,Y 327.039,Z 228.73,A -85,B 0,C 180,E1 -14941.232,E2 -14941.232} C_VEL
LIN {X 0,Y 326.753,Z 228.755,A -85,B 0,C 180,E1 -14943.7,E2 -14943.7} C_VEL
LIN {X 0,Y 326.949,Z 228.752,A -85,B 0,C 180,E1 -14946.642,E2 -14946.642} C_VEL
LIN {X 0,Y 326.797,Z 228.75,A -85,B 0,C 180,E1 -14949.907,E2 -14949.907} C_VEL
LIN {X 0,Y 326.751,Z 228.78,A -85,B 0,C 180,E1 -14953.686,E2 -14953.686} C_VEL
LIN {X 0,Y 326.655,Z 228.773,A -85,B 0,C 180,E1 -14957.531,E2 -14957.531} C_VEL
LIN {X 0,Y 326.647,Z 228.796,A -85,B 0,C 180,E1 -14960.136,E2 -14960.136} C_VEL
LIN {X 0,Y 326.645,Z 228.78,A -85,B 0,C 180,E1 -14964.13,E2 -14964.13} C_VEL
LIN {X 0,Y 326.676,Z 228.793,A -85,B 0,C 180,E1 -14966.859,E2 -14966.859} C_VEL
LIN {X 0,Y 326.628,Z 228.794,A -85,B 0,C 180,E1 -14970.611,E2 -14970.611} C_VEL
LIN {X 0,Y 326.601,Z 228.791,A -85,B 0,C 180,E1 -14974.021,E2 -14974.021} C_VEL
LIN {X 0,Y 326.623,Z 228.798,A -85,B 0,C 180,E1 -14977.24,E2 -14977.24} C_VEL
LIN {X 0,Y 326.573,Z 228.804,A -85,B 0,C 180,E1 -14981.133,E2 -14981.133} C_VEL
LIN {X 0,Y 326.525,Z 228.808,A -85,B 0,C 180,E1 -14984.745,E2 -14984.745} C_VEL
LIN {X 0,Y 326.573,Z 228.804,A -85,B 0,C 180,E1 -14988.156,E2 -14988.156} C_VEL
LIN {X 0,Y 326.601,Z 228.799,A -85,B 0,C 180,E1 -14989.352,E2 -14989.352} C_VEL
LIN {X 0,Y 327.652,Z 231.706,A -85,B 0,C 180,E1 -14989.544,E2 -14989.544} C_VEL
LIN {X 0,Y 332.476,Z 240.295,A -85,B 0,C 180,E1 -14990.257,E2 -14990.257} C_VEL
LIN {X 0,Y 339.372,Z 254.367,A -85,B 0,C 180,E1 -14991.274,E2 -14991.274} C_VEL
LIN {X 0,Y 341.244,Z 259.025,A -85,B 0,C 180,E1 -14991.56,E2 -14991.56} C_VEL
LIN {X 0,Y 339.061,Z 339.172,A -85,B 0,C 180,E1 -14993.285,E2 -14993.285} C_VEL
LIN {X 0,Y 338.406,Z 352.387,A -85,B 0,C 180,E1 -14993.788,E2 -14993.788} C_VEL
LIN {X 0,Y 337.552,Z 364.027,A -85,B 0,C 180,E1 -14994.456,E2 -14994.456} C_VEL
LIN {X 0,Y 336.401,Z 375.087,A -85,B 0,C 180,E1 -14995.3,E2 -14995.3} C_VEL
LIN {X 0,Y 335.025,Z 386.313,A -85,B 0,C 180,E1 -14996.409,E2 -14996.409} C_VEL
LIN {X 0,Y 333.39,Z 396.998,A -85,B 0,C 180,E1 -14997.734,E2 -14997.734} C_VEL
LIN {X 0,Y 331.927,Z 405.856,A -85,B 0,C 180,E1 -14999.108,E2 -14999.108} C_VEL
LIN {X 0,Y 330.467,Z 414.289,A -85,B 0,C 180,E1 -15000.718,E2 -15000.718} C_VEL
LIN {X 0,Y 328.932,Z 422.461,A -85,B 0,C 180,E1 -15002.655,E2 -15002.655} C_VEL
LIN {X 0,Y 327.716,Z 428.893,A -85,B 0,C 180,E1 -15004.603,E2 -15004.603} C_VEL
LIN {X 0,Y 326.747,Z 433.911,A -85,B 0,C 180,E1 -15006.554,E2 -15006.554} C_VEL
LIN {X 0,Y 326.004,Z 437.698,A -85,B 0,C 180,E1 -15008.502,E2 -15008.502} C_VEL
LIN {X 0,Y 325.602,Z 439.619,A -85,B 0,C 180,E1 -15009.798,E2 -15009.798} C_VEL
LIN {X 0,Y 325.161,Z 441.801,A -85,B 0,C 180,E1 -15011.994,E2 -15011.994} C_VEL
LIN {X 0,Y 324.926,Z 442.621,A -85,B 0,C 180,E1 -15013.671,E2 -15013.671} C_VEL
LIN {X 0,Y 324.82,Z 442.766,A -85,B 0,C 180,E1 -15014.953,E2 -15014.953} C_VEL
LIN {X 0,Y 324.847,Z 442.237,A -85,B 0,C 180,E1 -15016.799,E2 -15016.799} C_VEL
LIN {X 0,Y 324.899,Z 440.688,A -85,B 0,C 180,E1 -15018.775,E2 -15018.775} C_VEL
LIN {X 0,Y 325.02,Z 439.129,A -85,B 0,C 180,E1 -15020.04,E2 -15020.04} C_VEL
LIN {X 0,Y 325.302,Z 435.99,A -85,B 0,C 180,E1 -15021.929,E2 -15021.929} C_VEL
LIN {X 0,Y 325.709,Z 431.781,A -85,B 0,C 180,E1 -15023.808,E2 -15023.808} C_VEL
LIN {X 0,Y 326.264,Z 425.408,A -85,B 0,C 180,E1 -15025.987,E2 -15025.987} C_VEL
LIN {X 0,Y 326.979,Z 418.391,A -85,B 0,C 180,E1 -15027.846,E2 -15027.846} C_VEL
LIN {X 0,Y 327.958,Z 409.652,A -85,B 0,C 180,E1 -15029.694,E2 -15029.694} C_VEL
LIN {X 0,Y 328.957,Z 400.688,A -85,B 0,C 180,E1 -15031.226,E2 -15031.226} C_VEL
LIN {X 0,Y 330.052,Z 390.734,A -85,B 0,C 180,E1 -15032.595,E2 -15032.595} C_VEL
LIN {X 0,Y 331.165,Z 378.774,A -85,B 0,C 180,E1 -15033.905,E2 -15033.905} C_VEL
LIN {X 0,Y 331.959,Z 367.566,A -85,B 0,C 180,E1 -15034.859,E2 -15034.859} C_VEL
LIN {X 0,Y 332.705,Z 354.463,A -85,B 0,C 180,E1 -15035.684,E2 -15035.684} C_VEL
LIN {X 0,Y 333.245,Z 341.792,A -85,B 0,C 180,E1 -15036.23,E2 -15036.23} C_VEL
LIN {X 0,Y 333.79,Z 318.258,A -85,B 0,C 180,E1 -15036.779,E2 -15036.779} C_VEL
LIN {X 0,Y 334.888,Z 256.371,A -85,B 0,C 180,E1 -15038.097,E2 -15038.097} C_VEL
LIN {X 0,Y 332.998,Z 245.3,A -85,B 0,C 180,E1 -15038.453,E2 -15038.453} C_VEL
LIN {X 0,Y 326.834,Z 228.772,A -85,B 0,C 180,E1 -15039.213,E2 -15039.213} C_VEL
LIN {X 0,Y 326.741,Z 228.787,A -85,B 0,C 180,E1 -15042.422,E2 -15042.422} C_VEL
LIN {X 0,Y 326.76,Z 228.781,A -85,B 0,C 180,E1 -15044.959,E2 -15044.959} C_VEL
LIN {X 0,Y 326.739,Z 228.783,A -85,B 0,C 180,E1 -15048.839,E2 -15048.839} C_VEL
LIN {X 0,Y 326.599,Z 228.8,A -85,B 0,C 180,E1 -15052.79,E2 -15052.79} C_VEL
LIN {X 0,Y 326.604,Z 228.799,A -85,B 0,C 180,E1 -15056.866,E2 -15056.866} C_VEL
LIN {X 0,Y 326.579,Z 228.801,A -85,B 0,C 180,E1 -15061.098,E2 -15061.098} C_VEL
LIN {X 0,Y 326.591,Z 228.799,A -85,B 0,C 180,E1 -15062.259,E2 -15062.259} C_VEL
LIN {X 0,Y 325.984,Z 228.88,A -85,B 0,C 180,E1 -15063.289,E2 -15063.289} C_VEL
LIN {X 0,Y 323.165,Z 229.238,A -85,B 0,C 180,E1 -15064.965,E2 -15064.965} C_VEL
LIN {X 0,Y 320.721,Z 229.542,A -85,B 0,C 180,E1 -15066.322,E2 -15066.322} C_VEL
LIN {X 0,Y 319.643,Z 229.672,A -85,B 0,C 180,E1 -15067.374,E2 -15067.374} C_VEL
LIN {X 0,Y 319.542,Z 229.682,A -85,B 0,C 180,E1 -15067.73,E2 -15067.73} C_VEL
LIN {X 0,Y 319.509,Z 229.686,A -85,B 0,C 180,E1 -15071.593,E2 -15071.593} C_VEL
LIN {X 0,Y 319.491,Z 229.684,A -85,B 0,C 180,E1 -15074.744,E2 -15074.744} C_VEL
LIN {X 0,Y 319.556,Z 229.679,A -85,B 0,C 180,E1 -15077.016,E2 -15077.016} C_VEL
LIN {X 0,Y 319.521,Z 229.679,A -85,B 0,C 180,E1 -15080.366,E2 -15080.366} C_VEL
LIN {X 0,Y 319.56,Z 229.677,A -85,B 0,C 180,E1 -15083.572,E2 -15083.572} C_VEL
LIN {X 0,Y 319.583,Z 229.676,A -85,B 0,C 180,E1 -15086.687,E2 -15086.687} C_VEL
LIN {X 0,Y 319.558,Z 229.675,A -85,B 0,C 180,E1 -15089.613,E2 -15089.613} C_VEL
LIN {X 0,Y 319.54,Z 229.676,A -85,B 0,C 180,E1 -15092.491,E2 -15092.491} C_VEL
LIN {X 0,Y 319.638,Z 229.735,A -85,B 0,C 180,E1 -15095.825,E2 -15095.825} C_VEL
LIN {X 0,Y 320.138,Z 232.419,A -85,B 0,C 180,E1 -15096.653,E2 -15096.653} C_VEL
LIN {X 0,Y 325.089,Z 251.465,A -85,B 0,C 180,E1 -15097.481,E2 -15097.481} C_VEL
LIN {X 0,Y 326.244,Z 259.05,A -85,B 0,C 180,E1 -15097.772,E2 -15097.772} C_VEL
LIN {X 0,Y 323.577,Z 341.096,A -85,B 0,C 180,E1 -15100.368,E2 -15100.368} C_VEL
LIN {X 0,Y 323.139,Z 354.639,A -85,B 0,C 180,E1 -15101.041,E2 -15101.041} C_VEL
LIN {X 0,Y 322.561,Z 367.234,A -85,B 0,C 180,E1 -15101.911,E2 -15101.911} C_VEL
LIN {X 0,Y 321.746,Z 379.48,A -85,B 0,C 180,E1 -15103.013,E2 -15103.013} C_VEL
LIN {X 0,Y 320.948,Z 390.676,A -85,B 0,C 180,E1 -15104.277,E2 -15104.277} C_VEL
LIN {X 0,Y 320.26,Z 401.9,A -85,B 0,C 180,E1 -15105.869,E2 -15105.869} C_VEL
LIN {X 0,Y 319.497,Z 411.873,A -85,B 0,C 180,E1 -15107.615,E2 -15107.615} C_VEL
LIN {X 0,Y 318.891,Z 420.602,A -85,B 0,C 180,E1 -15109.524,E2 -15109.524} C_VEL
LIN {X 0,Y 318.453,Z 427.643,A -85,B 0,C 180,E1 -15111.433,E2 -15111.433} C_VEL
LIN {X 0,Y 318.214,Z 432.366,A -85,B 0,C 180,E1 -15113.023,E2 -15113.023} C_VEL
LIN {X 0,Y 318.04,Z 436.887,A -85,B 0,C 180,E1 -15114.929,E2 -15114.929} C_VEL
LIN {X 0,Y 318.016,Z 439.248,A -85,B 0,C 180,E1 -15116.198,E2 -15116.198} C_VEL
LIN {X 0,Y 317.916,Z 441.119,A -85,B 0,C 180,E1 -15117.466,E2 -15117.466} C_VEL
LIN {X 0,Y 317.899,Z 442.565,A -85,B 0,C 180,E1 -15118.733,E2 -15118.733} C_VEL
LIN {X 0,Y 317.981,Z 443.555,A -85,B 0,C 180,E1 -15120,E2 -15120} C_VEL
LIN {X 0,Y 318.133,Z 444.086,A -85,B 0,C 180,E1 -15121.266,E2 -15121.266} C_VEL
LIN {X 0,Y 318.345,Z 444.205,A -85,B 0,C 180,E1 -15122.53,E2 -15122.53} C_VEL
LIN {X 0,Y 318.668,Z 443.906,A -85,B 0,C 180,E1 -15123.793,E2 -15123.793} C_VEL
LIN {X 0,Y 319.029,Z 443.14,A -85,B 0,C 180,E1 -15125.055,E2 -15125.055} C_VEL
LIN {X 0,Y 319.308,Z 441.973,A -85,B 0,C 180,E1 -15126.318,E2 -15126.318} C_VEL
LIN {X 0,Y 319.492,Z 440.412,A -85,B 0,C 180,E1 -15127.584,E2 -15127.584} C_VEL
LIN {X 0,Y 320.819,Z 436.692,A -85,B 0,C 180,E1 -15129.664,E2 -15129.664} C_VEL
LIN {X 0,Y 321.848,Z 432.742,A -85,B 0,C 180,E1 -15131.334,E2 -15131.334} C_VEL
LIN {X 0,Y 323.601,Z 426.082,A -85,B 0,C 180,E1 -15133.501,E2 -15133.501} C_VEL
LIN {X 0,Y 325.405,Z 418.849,A -85,B 0,C 180,E1 -15135.341,E2 -15135.341} C_VEL
LIN {X 0,Y 327.468,Z 409.935,A -85,B 0,C 180,E1 -15137.163,E2 -15137.163} C_VEL
LIN {X 0,Y 329.902,Z 398.761,A -85,B 0,C 180,E1 -15138.958,E2 -15138.958} C_VEL
LIN {X 0,Y 332.165,Z 387.053,A -85,B 0,C 180,E1 -15140.433,E2 -15140.433} C_VEL
LIN {X 0,Y 334.079,Z 375.5,A -85,B 0,C 180,E1 -15141.601,E2 -15141.601} C_VEL
LIN {X 0,Y 335.924,Z 362.262,A -85,B 0,C 180,E1 -15142.628,E2 -15142.628} C_VEL
LIN {X 0,Y 337.39,Z 349.066,A -85,B 0,C 180,E1 -15143.396,E2 -15143.396} C_VEL
LIN {X 0,Y 338.858,Z 331.404,A -85,B 0,C 180,E1 -15144.099,E2 -15144.099} C_VEL
LIN {X 0,Y 344.081,Z 275.486,A -85,B 0,C 180,E1 -15146.131,E2 -15146.131} C_VEL
LIN {X 0,Y 339.72,Z 266.553,A -85,B 0,C 180,E1 -15147.483,E2 -15147.483} C_VEL
LIN {X 0,Y 335.351,Z 259.102,A -85,B 0,C 180,E1 -15148.909,E2 -15148.909} C_VEL
LIN {X 0,Y 333.103,Z 255.69,A -85,B 0,C 180,E1 -15149.695,E2 -15149.695} C_VEL
LIN {X 0,Y 330.736,Z 252.19,A -85,B 0,C 180,E1 -15150.581,E2 -15150.581} C_VEL
LIN {X 0,Y 327.939,Z 248.325,A -85,B 0,C 180,E1 -15151.714,E2 -15151.714} C_VEL
LIN {X 0,Y 324.343,Z 243.91,A -85,B 0,C 180,E1 -15153.329,E2 -15153.329} C_VEL
LIN {X 0,Y 323.827,Z 242.899,A -85,B 0,C 180,E1 -15153.639,E2 -15153.639} C_VEL
LIN {X 0,Y 323.225,Z 240.841,A -85,B 0,C 180,E1 -15156.436,E2 -15156.436} C_VEL
LIN {X 0,Y 322.893,Z 239.786,A -85,B 0,C 180,E1 -15159.139,E2 -15159.139} C_VEL
LIN {X 0,Y 322.818,Z 239.607,A -85,B 0,C 180,E1 -15162.446,E2 -15162.446} C_VEL
LIN {X 0,Y 323.282,Z 240.769,A -85,B 0,C 180,E1 -15165.918,E2 -15165.918} C_VEL
LIN {X 0,Y 323.624,Z 241.967,A -85,B 0,C 180,E1 -15167.683,E2 -15167.683} C_VEL
LIN {X 0,Y 324.68,Z 245.463,A -85,B 0,C 180,E1 -15171.192,E2 -15171.192} C_VEL
LIN {X 0,Y 325.598,Z 248.516,A -85,B 0,C 180,E1 -15173.439,E2 -15173.439} C_VEL
LIN {X 0,Y 326.894,Z 253.639,A -85,B 0,C 180,E1 -15176.427,E2 -15176.427} C_VEL
LIN {X 0,Y 329.925,Z 259.222,A -85,B 0,C 180,E1 -15177.758,E2 -15177.758} C_VEL
LIN {X 0,Y 331.106,Z 261.191,A -85,B 0,C 180,E1 -15178.212,E2 -15178.212} C_VEL
LIN {X 0,Y 334.286,Z 267.373,A -85,B 0,C 180,E1 -15179.423,E2 -15179.423} C_VEL
LIN {X 0,Y 337.103,Z 273.442,A -85,B 0,C 180,E1 -15180.431,E2 -15180.431} C_VEL
LIN {X 0,Y 337.987,Z 276.068,A -85,B 0,C 180,E1 -15180.771,E2 -15180.771} C_VEL
LIN {X 0,Y 340.244,Z 288.941,A -85,B 0,C 180,E1 -15181.956,E2 -15181.956} C_VEL
LIN {X 0,Y 341.723,Z 301.083,A -85,B 0,C 180,E1 -15182.875,E2 -15182.875} C_VEL
LIN {X 0,Y 341.973,Z 306.4,A -85,B 0,C 180,E1 -15183.193,E2 -15183.193} C_VEL
LIN {X 0,Y 336.521,Z 368.972,A -85,B 0,C 180,E1 -15185.475,E2 -15185.475} C_VEL
LIN {X 0,Y 334.746,Z 382.451,A -85,B 0,C 180,E1 -15186.161,E2 -15186.161} C_VEL
LIN {X 0,Y 332.615,Z 396.315,A -85,B 0,C 180,E1 -15187.153,E2 -15187.153} C_VEL
LIN {X 0,Y 330.295,Z 408.794,A -85,B 0,C 180,E1 -15188.301,E2 -15188.301} C_VEL
LIN {X 0,Y 328.083,Z 420.076,A -85,B 0,C 180,E1 -15189.628,E2 -15189.628} C_VEL
LIN {X 0,Y 325.904,Z 430.432,A -85,B 0,C 180,E1 -15191.126,E2 -15191.126} C_VEL
LIN {X 0,Y 323.58,Z 440.616,A -85,B 0,C 180,E1 -15192.96,E2 -15192.96} C_VEL
LIN {X 0,Y 321.927,Z 448.815,A -85,B 0,C 180,E1 -15194.811,E2 -15194.811} C_VEL
LIN {X 0,Y 320.43,Z 455.54,A -85,B 0,C 180,E1 -15196.684,E2 -15196.684} C_VEL
LIN {X 0,Y 319.343,Z 460.952,A -85,B 0,C 180,E1 -15198.575,E2 -15198.575} C_VEL
LIN {X 0,Y 318.565,Z 465.22,A -85,B 0,C 180,E1 -15200.475,E2 -15200.475} C_VEL
LIN {X 0,Y 318.066,Z 468.418,A -85,B 0,C 180,E1 -15202.38,E2 -15202.38} C_VEL
LIN {X 0,Y 317.845,Z 470.604,A -85,B 0,C 180,E1 -15204.277,E2 -15204.277} C_VEL
LIN {X 0,Y 317.837,Z 471.829,A -85,B 0,C 180,E1 -15206.195,E2 -15206.195} C_VEL
LIN {X 0,Y 317.814,Z 472.067,A -85,B 0,C 180,E1 -15207.464,E2 -15207.464} C_VEL
LIN {X 0,Y 317.918,Z 471.881,A -85,B 0,C 180,E1 -15208.732,E2 -15208.732} C_VEL
LIN {X 0,Y 318.121,Z 471.276,A -85,B 0,C 180,E1 -15209.999,E2 -15209.999} C_VEL
LIN {X 0,Y 317.896,Z 470.892,A -85,B 0,C 180,E1 -15212.533,E2 -15212.533} C_VEL
LIN {X 0,Y 317.873,Z 470.26,A -85,B 0,C 180,E1 -15213.802,E2 -15213.802} C_VEL
LIN {X 0,Y 317.898,Z 468.432,A -85,B 0,C 180,E1 -15215.819,E2 -15215.819} C_VEL
LIN {X 0,Y 318.16,Z 464.836,A -85,B 0,C 180,E1 -15218.254,E2 -15218.254} C_VEL
LIN {X 0,Y 318.63,Z 460.829,A -85,B 0,C 180,E1 -15220.162,E2 -15220.162} C_VEL
LIN {X 0,Y 319.538,Z 454.664,A -85,B 0,C 180,E1 -15222.381,E2 -15222.381} C_VEL
LIN {X 0,Y 320.833,Z 447.957,A -85,B 0,C 180,E1 -15224.265,E2 -15224.265} C_VEL
LIN {X 0,Y 322.133,Z 439.942,A -85,B 0,C 180,E1 -15226.088,E2 -15226.088} C_VEL
LIN {X 0,Y 323.714,Z 431.098,A -85,B 0,C 180,E1 -15227.693,E2 -15227.693} C_VEL
LIN {X 0,Y 325.567,Z 420.569,A -85,B 0,C 180,E1 -15229.219,E2 -15229.219} C_VEL
LIN {X 0,Y 327.231,Z 410.125,A -85,B 0,C 180,E1 -15230.425,E2 -15230.425} C_VEL
LIN {X 0,Y 328.782,Z 398.503,A -85,B 0,C 180,E1 -15231.471,E2 -15231.471} C_VEL
LIN {X 0,Y 330.189,Z 386.452,A -85,B 0,C 180,E1 -15232.279,E2 -15232.279} C_VEL
LIN {X 0,Y 331.39,Z 373.26,A -85,B 0,C 180,E1 -15232.892,E2 -15232.892} C_VEL
LIN {X 0,Y 331.929,Z 358.589,A -85,B 0,C 180,E1 -15233.306,E2 -15233.306} C_VEL
LIN {X 0,Y 333.328,Z 302.754,A -85,B 0,C 180,E1 -15234.538,E2 -15234.538} C_VEL
LIN {X 0,Y 330.325,Z 280.809,A -85,B 0,C 180,E1 -15235.368,E2 -15235.368} C_VEL
LIN {X 0,Y 325.107,Z 251.595,A -85,B 0,C 180,E1 -15236.632,E2 -15236.632} C_VEL
LIN {X 0,Y 323.424,Z 246.874,A -85,B 0,C 180,E1 -15236.936,E2 -15236.936} C_VEL
LIN {X 0,Y 322.295,Z 243.113,A -85,B 0,C 180,E1 -15237.216,E2 -15237.216} C_VEL
LIN {X 0,Y 319.618,Z 229.672,A -85,B 0,C 180,E1 -15240.922,E2 -15240.922} C_VEL
LIN {X 0,Y 319.555,Z 229.653,A -85,B 0,C 180,E1 -15244.875,E2 -15244.875} C_VEL
LIN {X 0,Y 319.518,Z 229.678,A -85,B 0,C 180,E1 -15248.014,E2 -15248.014} C_VEL
LIN {X 0,Y 319.499,Z 229.686,A -85,B 0,C 180,E1 -15251.592,E2 -15251.592} C_VEL
LIN {X 0,Y 319.481,Z 229.685,A -85,B 0,C 180,E1 -15254.742,E2 -15254.742} C_VEL
LIN {X 0,Y 319.545,Z 229.674,A -85,B 0,C 180,E1 -15257.015,E2 -15257.015} C_VEL
LIN {X 0,Y 319.537,Z 229.679,A -85,B 0,C 180,E1 -15260.37,E2 -15260.37} C_VEL
LIN {X 0,Y 319.571,Z 229.654,A -85,B 0,C 180,E1 -15264.456,E2 -15264.456} C_VEL
LIN {X 0,Y 319.516,Z 229.678,A -85,B 0,C 180,E1 -15268.137,E2 -15268.137} C_VEL
LIN {X 0,Y 319.536,Z 229.658,A -85,B 0,C 180,E1 -15271.612,E2 -15271.612} C_VEL
LIN {X 0,Y 319.562,Z 229.669,A -85,B 0,C 180,E1 -15275.301,E2 -15275.301} C_VEL
LIN {X 0,Y 319.556,Z 229.646,A -85,B 0,C 180,E1 -15278.045,E2 -15278.045} C_VEL
LIN {X 0,Y 319.605,Z 229.67,A -85,B 0,C 180,E1 -15282.07,E2 -15282.07} C_VEL
LIN {X 0,Y 319.721,Z 229.627,A -85,B 0,C 180,E1 -15286.008,E2 -15286.008} C_VEL
LIN {X 0,Y 319.726,Z 229.657,A -85,B 0,C 180,E1 -15289.872,E2 -15289.872} C_VEL
LIN {X 0,Y 319.887,Z 229.612,A -85,B 0,C 180,E1 -15293.694,E2 -15293.694} C_VEL
LIN {X 0,Y 319.967,Z 229.621,A -85,B 0,C 180,E1 -15297.482,E2 -15297.482} C_VEL
LIN {X 0,Y 320.006,Z 229.604,A -85,B 0,C 180,E1 -15301.259,E2 -15301.259} C_VEL
LIN {X 0,Y 319.933,Z 229.63,A -85,B 0,C 180,E1 -15306.306,E2 -15306.306} C_VEL
LIN {X 0,Y 319.829,Z 229.629,A -85,B 0,C 180,E1 -15308.849,E2 -15308.849} C_VEL
LIN {X 0,Y 319.674,Z 229.658,A -85,B 0,C 180,E1 -15312.701,E2 -15312.701} C_VEL
LIN {X 0,Y 319.671,Z 229.66,A -85,B 0,C 180,E1 -15315.297,E2 -15315.297} C_VEL
LIN {X 0,Y 319.626,Z 229.662,A -85,B 0,C 180,E1 -15319.258,E2 -15319.258} C_VEL
LIN {X 0,Y 319.563,Z 229.662,A -85,B 0,C 180,E1 -15323.32,E2 -15323.32} C_VEL
LIN {X 0,Y 319.628,Z 229.671,A -85,B 0,C 180,E1 -15326.089,E2 -15326.089} C_VEL
LIN {X 0,Y 319.573,Z 229.665,A -85,B 0,C 180,E1 -15328.936,E2 -15328.936} C_VEL
LIN {X 0,Y 319.525,Z 229.685,A -85,B 0,C 180,E1 -15331.863,E2 -15331.863} C_VEL
LIN {X 0,Y 319.575,Z 229.677,A -85,B 0,C 180,E1 -15335.544,E2 -15335.544} C_VEL
LIN {X 0,Y 319.553,Z 229.673,A -85,B 0,C 180,E1 -15338.012,E2 -15338.012} C_VEL
LIN {X 0,Y 319.521,Z 229.678,A -85,B 0,C 180,E1 -15341.599,E2 -15341.599} C_VEL
LIN {X 0,Y 319.486,Z 229.685,A -85,B 0,C 180,E1 -15344.744,E2 -15344.744} C_VEL
LIN {X 0,Y 319.537,Z 229.683,A -85,B 0,C 180,E1 -15348.505,E2 -15348.505} C_VEL
LIN {X 0,Y 319.549,Z 229.763,A -85,B 0,C 180,E1 -15348.607,E2 -15348.607} C_VEL
LIN {X 0,Y 320.539,Z 232.544,A -85,B 0,C 180,E1 -15348.792,E2 -15348.792} C_VEL
LIN {X 0,Y 325.092,Z 240.402,A -85,B 0,C 180,E1 -15349.493,E2 -15349.493} C_VEL
LIN {X 0,Y 333.255,Z 256.507,A -85,B 0,C 180,E1 -15350.735,E2 -15350.735} C_VEL
LIN {X 0,Y 335.011,Z 260.81,A -85,B 0,C 180,E1 -15351.013,E2 -15351.013} C_VEL
LIN {X 0,Y 332.737,Z 340.101,A -85,B 0,C 180,E1 -15352.754,E2 -15352.754} C_VEL
LIN {X 0,Y 332.022,Z 353.365,A -85,B 0,C 180,E1 -15353.277,E2 -15353.277} C_VEL
LIN {X 0,Y 331.084,Z 365.381,A -85,B 0,C 180,E1 -15353.999,E2 -15353.999} C_VEL
LIN {X 0,Y 329.612,Z 378.269,A -85,B 0,C 180,E1 -15355.04,E2 -15355.04} C_VEL
LIN {X 0,Y 328.217,Z 388.908,A -85,B 0,C 180,E1 -15356.172,E2 -15356.172} C_VEL
LIN {X 0,Y 326.387,Z 399.735,A -85,B 0,C 180,E1 -15357.615,E2 -15357.615} C_VEL
LIN {X 0,Y 324.865,Z 408.548,A -85,B 0,C 180,E1 -15359.085,E2 -15359.085} C_VEL
LIN {X 0,Y 323.33,Z 416.861,A -85,B 0,C 180,E1 -15360.793,E2 -15360.793} C_VEL
LIN {X 0,Y 321.845,Z 424.295,A -85,B 0,C 180,E1 -15362.707,E2 -15362.707} C_VEL
LIN {X 0,Y 320.591,Z 430.416,A -85,B 0,C 180,E1 -15364.694,E2 -15364.694} C_VEL
LIN {X 0,Y 319.62,Z 435.17,A -85,B 0,C 180,E1 -15366.686,E2 -15366.686} C_VEL
LIN {X 0,Y 319.088,Z 437.643,A -85,B 0,C 180,E1 -15368.013,E2 -15368.013} C_VEL
LIN {X 0,Y 318.641,Z 439.625,A -85,B 0,C 180,E1 -15369.337,E2 -15369.337} C_VEL
LIN {X 0,Y 318.298,Z 441.167,A -85,B 0,C 180,E1 -15370.66,E2 -15370.66} C_VEL
LIN {X 0,Y 318.085,Z 442.22,A -85,B 0,C 180,E1 -15371.983,E2 -15371.983} C_VEL
LIN {X 0,Y 317.878,Z 442.857,A -85,B 0,C 180,E1 -15373.298,E2 -15373.298} C_VEL
LIN {X 0,Y 317.753,Z 443.093,A -85,B 0,C 180,E1 -15374.61,E2 -15374.61} C_VEL
LIN {X 0,Y 317.758,Z 442.567,A -85,B 0,C 180,E1 -15376.7,E2 -15376.7} C_VEL
LIN {X 0,Y 317.802,Z 441.218,A -85,B 0,C 180,E1 -15378.521,E2 -15378.521} C_VEL
LIN {X 0,Y 317.892,Z 439.759,A -85,B 0,C 180,E1 -15379.814,E2 -15379.814} C_VEL
LIN {X 0,Y 318.184,Z 436.737,A -85,B 0,C 180,E1 -15381.747,E2 -15381.747} C_VEL
LIN {X 0,Y 318.595,Z 432.653,A -85,B 0,C 180,E1 -15383.669,E2 -15383.669} C_VEL
LIN {X 0,Y 319.147,Z 426.417,A -85,B 0,C 180,E1 -15385.897,E2 -15385.897} C_VEL
LIN {X 0,Y 319.853,Z 419.618,A -85,B 0,C 180,E1 -15387.798,E2 -15387.798} C_VEL
LIN {X 0,Y 320.849,Z 411.067,A -85,B 0,C 180,E1 -15389.688,E2 -15389.688} C_VEL
LIN {X 0,Y 321.872,Z 402.317,A -85,B 0,C 180,E1 -15391.253,E2 -15391.253} C_VEL
LIN {X 0,Y 322.96,Z 392.728,A -85,B 0,C 180,E1 -15392.652,E2 -15392.652} C_VEL
LIN {X 0,Y 324.042,Z 382.049,A -85,B 0,C 180,E1 -15393.9,E2 -15393.9} C_VEL
LIN {X 0,Y 324.93,Z 370.506,A -85,B 0,C 180,E1 -15394.965,E2 -15394.965} C_VEL
LIN {X 0,Y 325.746,Z 358.486,A -85,B 0,C 180,E1 -15395.806,E2 -15395.806} C_VEL
LIN {X 0,Y 326.307,Z 346.183,A -85,B 0,C 180,E1 -15396.416,E2 -15396.416} C_VEL
LIN {X 0,Y 326.678,Z 332.41,A -85,B 0,C 180,E1 -15396.836,E2 -15396.836} C_VEL
LIN {X 0,Y 328.229,Z 257.709,A -85,B 0,C 180,E1 -15398.448,E2 -15398.448} C_VEL
LIN {X 0,Y 326.366,Z 247.112,A -85,B 0,C 180,E1 -15398.801,E2 -15398.801} C_VEL
LIN {X 0,Y 319.887,Z 230.437,A -85,B 0,C 180,E1 -15399.586,E2 -15399.586} C_VEL
LIN {X 0,Y 319.744,Z 229.655,A -85,B 0,C 180,E1 -15399.634,E2 -15399.634} C_VEL
LIN {X 0,Y 319.688,Z 229.665,A -85,B 0,C 180,E1 -15402.701,E2 -15402.701} C_VEL
LIN {X 0,Y 319.706,Z 229.659,A -85,B 0,C 180,E1 -15405.297,E2 -15405.297} C_VEL
LIN {X 0,Y 319.658,Z 229.664,A -85,B 0,C 180,E1 -15409.257,E2 -15409.257} C_VEL
LIN {X 0,Y 319.548,Z 229.678,A -85,B 0,C 180,E1 -15413.322,E2 -15413.322} C_VEL
LIN {X 0,Y 319.556,Z 229.681,A -85,B 0,C 180,E1 -15416.096,E2 -15416.096} C_VEL
LIN {X 0,Y 319.531,Z 229.68,A -85,B 0,C 180,E1 -15418.941,E2 -15418.941} C_VEL
LIN {X 0,Y 319.525,Z 229.682,A -85,B 0,C 180,E1 -15422.26,E2 -15422.26} C_VEL
LIN {X 0,Y 319.584,Z 229.677,A -85,B 0,C 180,E1 -15425.543,E2 -15425.543} C_VEL
LIN {X 0,Y 319.542,Z 229.682,A -85,B 0,C 180,E1 -15427.73,E2 -15427.73} C_VEL
LIN {X 0,Y 318.834,Z 229.768,A -85,B 0,C 180,E1 -15428.781,E2 -15428.781} C_VEL
LIN {X 0,Y 315.954,Z 230.125,A -85,B 0,C 180,E1 -15430.491,E2 -15430.491} C_VEL
LIN {X 0,Y 313.542,Z 230.426,A -85,B 0,C 180,E1 -15431.878,E2 -15431.878} C_VEL
LIN {X 0,Y 312.517,Z 230.552,A -85,B 0,C 180,E1 -15432.951,E2 -15432.951} C_VEL
LIN {X 0,Y 312.438,Z 230.559,A -85,B 0,C 180,E1 -15433.315,E2 -15433.315} C_VEL
LIN {X 0,Y 312.462,Z 230.561,A -85,B 0,C 180,E1 -15436.036,E2 -15436.036} C_VEL
LIN {X 0,Y 312.461,Z 230.559,A -85,B 0,C 180,E1 -15439.886,E2 -15439.886} C_VEL
LIN {X 0,Y 312.538,Z 230.55,A -85,B 0,C 180,E1 -15444.052,E2 -15444.052} C_VEL
LIN {X 0,Y 312.505,Z 230.557,A -85,B 0,C 180,E1 -15447.333,E2 -15447.333} C_VEL
LIN {X 0,Y 312.503,Z 230.551,A -85,B 0,C 180,E1 -15451.295,E2 -15451.295} C_VEL
LIN {X 0,Y 312.591,Z 230.563,A -85,B 0,C 180,E1 -15455.687,E2 -15455.687} C_VEL
LIN {X 0,Y 312.992,Z 232.732,A -85,B 0,C 180,E1 -15456.369,E2 -15456.369} C_VEL
LIN {X 0,Y 318.195,Z 252.787,A -85,B 0,C 180,E1 -15457.257,E2 -15457.257} C_VEL
LIN {X 0,Y 319.273,Z 260.06,A -85,B 0,C 180,E1 -15457.543,E2 -15457.543} C_VEL
LIN {X 0,Y 316.551,Z 341.517,A -85,B 0,C 180,E1 -15460.209,E2 -15460.209} C_VEL
LIN {X 0,Y 316.058,Z 355.628,A -85,B 0,C 180,E1 -15460.937,E2 -15460.937} C_VEL
LIN {X 0,Y 315.478,Z 367.988,A -85,B 0,C 180,E1 -15461.827,E2 -15461.827} C_VEL
LIN {X 0,Y 314.66,Z 380.129,A -85,B 0,C 180,E1 -15462.953,E2 -15462.953} C_VEL
LIN {X 0,Y 313.86,Z 391.375,A -85,B 0,C 180,E1 -15464.263,E2 -15464.263} C_VEL
LIN {X 0,Y 313.121,Z 402.443,A -85,B 0,C 180,E1 -15465.872,E2 -15465.872} C_VEL
LIN {X 0,Y 312.358,Z 412.377,A -85,B 0,C 180,E1 -15467.658,E2 -15467.658} C_VEL
LIN {X 0,Y 311.763,Z 421.082,A -85,B 0,C 180,E1 -15469.61,E2 -15469.61} C_VEL
LIN {X 0,Y 311.329,Z 428.1,A -85,B 0,C 180,E1 -15471.562,E2 -15471.562} C_VEL
LIN {X 0,Y 311.048,Z 433.651,A -85,B 0,C 180,E1 -15473.513,E2 -15473.513} C_VEL
LIN {X 0,Y 310.946,Z 437.951,A -85,B 0,C 180,E1 -15475.462,E2 -15475.462} C_VEL
LIN {X 0,Y 310.835,Z 441.12,A -85,B 0,C 180,E1 -15477.408,E2 -15477.408} C_VEL
LIN {X 0,Y 310.807,Z 442.644,A -85,B 0,C 180,E1 -15478.704,E2 -15478.704} C_VEL
LIN {X 0,Y 310.883,Z 443.751,A -85,B 0,C 180,E1 -15480,E2 -15480} C_VEL
LIN {X 0,Y 311.043,Z 444.41,A -85,B 0,C 180,E1 -15481.294,E2 -15481.294} C_VEL
LIN {X 0,Y 311.265,Z 444.613,A -85,B 0,C 180,E1 -15482.588,E2 -15482.588} C_VEL
LIN {X 0,Y 311.601,Z 444.402,A -85,B 0,C 180,E1 -15483.88,E2 -15483.88} C_VEL
LIN {X 0,Y 312.009,Z 443.78,A -85,B 0,C 180,E1 -15485.169,E2 -15485.169} C_VEL
LIN {X 0,Y 312.283,Z 442.717,A -85,B 0,C 180,E1 -15486.461,E2 -15486.461} C_VEL
LIN {X 0,Y 312.507,Z 441.249,A -85,B 0,C 180,E1 -15487.755,E2 -15487.755} C_VEL
LIN {X 0,Y 313.899,Z 437.713,A -85,B 0,C 180,E1 -15489.886,E2 -15489.886} C_VEL
LIN {X 0,Y 314.995,Z 433.962,A -85,B 0,C 180,E1 -15491.584,E2 -15491.584} C_VEL
LIN {X 0,Y 316.865,Z 427.613,A -85,B 0,C 180,E1 -15493.794,E2 -15493.794} C_VEL
LIN {X 0,Y 318.783,Z 420.648,A -85,B 0,C 180,E1 -15495.668,E2 -15495.668} C_VEL
LIN {X 0,Y 320.962,Z 412.073,A -85,B 0,C 180,E1 -15497.522,E2 -15497.522} C_VEL
LIN {X 0,Y 323.074,Z 403.348,A -85,B 0,C 180,E1 -15499.044,E2 -15499.044} C_VEL
LIN {X 0,Y 325.394,Z 392.72,A -85,B 0,C 180,E1 -15500.547,E2 -15500.547} C_VEL
LIN {X 0,Y 327.603,Z 380.996,A -85,B 0,C 180,E1 -15501.885,E2 -15501.885} C_VEL
LIN {X 0,Y 329.775,Z 367.906,A -85,B 0,C 180,E1 -15503.028,E2 -15503.028} C_VEL
LIN {X 0,Y 331.485,Z 354.438,A -85,B 0,C 180,E1 -15503.937,E2 -15503.937} C_VEL
LIN {X 0,Y 332.949,Z 339.8,A -85,B 0,C 180,E1 -15504.623,E2 -15504.623} C_VEL
LIN {X 0,Y 339.073,Z 278.513,A -85,B 0,C 180,E1 -15506.901,E2 -15506.901} C_VEL
LIN {X 0,Y 334.828,Z 269.739,A -85,B 0,C 180,E1 -15508.331,E2 -15508.331} C_VEL
LIN {X 0,Y 330.464,Z 262.341,A -85,B 0,C 180,E1 -15509.894,E2 -15509.894} C_VEL
LIN {X 0,Y 327.321,Z 257.803,A -85,B 0,C 180,E1 -15511.114,E2 -15511.114} C_VEL
LIN {X 0,Y 324.334,Z 253.562,A -85,B 0,C 180,E1 -15512.422,E2 -15512.422} C_VEL
LIN {X 0,Y 321.59,Z 249.932,A -85,B 0,C 180,E1 -15513.778,E2 -15513.778} C_VEL
LIN {X 0,Y 320.722,Z 248.888,A -85,B 0,C 180,E1 -15514.239,E2 -15514.239} C_VEL
LIN {X 0,Y 317.834,Z 245.589,A -85,B 0,C 180,E1 -15515.971,E2 -15515.971} C_VEL
LIN {X 0,Y 317.092,Z 244.377,A -85,B 0,C 180,E1 -15516.598,E2 -15516.598} C_VEL
LIN {X 0,Y 316.802,Z 243.446,A -85,B 0,C 180,E1 -15519.062,E2 -15519.062} C_VEL
LIN {X 0,Y 316.706,Z 243.19,A -85,B 0,C 180,E1 -15521.738,E2 -15521.738} C_VEL
LIN {X 0,Y 317.037,Z 244.09,A -85,B 0,C 180,E1 -15525.183,E2 -15525.183} C_VEL
LIN {X 0,Y 317.665,Z 246.239,A -85,B 0,C 180,E1 -15528.414,E2 -15528.414} C_VEL
LIN {X 0,Y 318.848,Z 249.889,A -85,B 0,C 180,E1 -15531.888,E2 -15531.888} C_VEL
LIN {X 0,Y 319.595,Z 252.601,A -85,B 0,C 180,E1 -15533.712,E2 -15533.712} C_VEL
LIN {X 0,Y 323.532,Z 259.134,A -85,B 0,C 180,E1 -15535.825,E2 -15535.825} C_VEL
LIN {X 0,Y 327.733,Z 266.829,A -85,B 0,C 180,E1 -15537.731,E2 -15537.731} C_VEL
LIN {X 0,Y 330.727,Z 272.928,A -85,B 0,C 180,E1 -15538.949,E2 -15538.949} C_VEL
LIN {X 0,Y 333.14,Z 278.348,A -85,B 0,C 180,E1 -15539.877,E2 -15539.877} C_VEL
LIN {X 0,Y 334.082,Z 282.537,A -85,B 0,C 180,E1 -15540.351,E2 -15540.351} C_VEL
LIN {X 0,Y 336.053,Z 296.262,A -85,B 0,C 180,E1 -15541.58,E2 -15541.58} C_VEL
LIN {X 0,Y 336.944,Z 306.845,A -85,B 0,C 180,E1 -15542.348,E2 -15542.348} C_VEL
LIN {X 0,Y 331.099,Z 368.903,A -85,B 0,C 180,E1 -15544.681,E2 -15544.681} C_VEL
LIN {X 0,Y 329.197,Z 382.466,A -85,B 0,C 180,E1 -15545.397,E2 -15545.397} C_VEL
LIN {X 0,Y 326.909,Z 396.151,A -85,B 0,C 180,E1 -15546.395,E2 -15546.395} C_VEL
LIN {X 0,Y 324.444,Z 408.476,A -85,B 0,C 180,E1 -15547.554,E2 -15547.554} C_VEL
LIN {X 0,Y 322.066,Z 419.678,A -85,B 0,C 180,E1 -15548.895,E2 -15548.895} C_VEL
LIN {X 0,Y 319.755,Z 429.976,A -85,B 0,C 180,E1 -15550.415,E2 -15550.415} C_VEL
LIN {X 0,Y 317.278,Z 440.076,A -85,B 0,C 180,E1 -15552.268,E2 -15552.268} C_VEL
LIN {X 0,Y 315.364,Z 448.319,A -85,B 0,C 180,E1 -15554.156,E2 -15554.156} C_VEL
LIN {X 0,Y 313.794,Z 455.035,A -85,B 0,C 180,E1 -15556.067,E2 -15556.067} C_VEL
LIN {X 0,Y 312.687,Z 459.648,A -85,B 0,C 180,E1 -15557.67,E2 -15557.67} C_VEL
LIN {X 0,Y 311.779,Z 464.111,A -85,B 0,C 180,E1 -15559.609,E2 -15559.609} C_VEL
LIN {X 0,Y 311.354,Z 466.467,A -85,B 0,C 180,E1 -15560.907,E2 -15560.907} C_VEL
LIN {X 0,Y 311.011,Z 468.372,A -85,B 0,C 180,E1 -15562.206,E2 -15562.206} C_VEL
LIN {X 0,Y 310.766,Z 470.534,A -85,B 0,C 180,E1 -15564.305,E2 -15564.305} C_VEL
LIN {X 0,Y 310.744,Z 471.5,A -85,B 0,C 180,E1 -15566.108,E2 -15566.108} C_VEL
LIN {X 0,Y 310.734,Z 471.664,A -85,B 0,C 180,E1 -15567.406,E2 -15567.406} C_VEL
LIN {X 0,Y 310.829,Z 471.411,A -85,B 0,C 180,E1 -15568.703,E2 -15568.703} C_VEL
LIN {X 0,Y 311.063,Z 470.715,A -85,B 0,C 180,E1 -15569.999,E2 -15569.999} C_VEL
LIN {X 0,Y 310.81,Z 470.611,A -85,B 0,C 180,E1 -15572.591,E2 -15572.591} C_VEL
LIN {X 0,Y 310.779,Z 470.001,A -85,B 0,C 180,E1 -15573.889,E2 -15573.889} C_VEL
LIN {X 0,Y 310.827,Z 467.607,A -85,B 0,C 180,E1 -15576.49,E2 -15576.49} C_VEL
LIN {X 0,Y 311.109,Z 464.679,A -85,B 0,C 180,E1 -15578.442,E2 -15578.442} C_VEL
LIN {X 0,Y 311.608,Z 460.725,A -85,B 0,C 180,E1 -15580.393,E2 -15580.393} C_VEL
LIN {X 0,Y 312.588,Z 454.644,A -85,B 0,C 180,E1 -15582.661,E2 -15582.661} C_VEL
LIN {X 0,Y 313.954,Z 448.002,A -85,B 0,C 180,E1 -15584.585,E2 -15584.585} C_VEL
LIN {X 0,Y 315.221,Z 440.557,A -85,B 0,C 180,E1 -15586.34,E2 -15586.34} C_VEL
LIN {X 0,Y 316.979,Z 431.356,A -85,B 0,C 180,E1 -15588.082,E2 -15588.082} C_VEL
LIN {X 0,Y 318.907,Z 420.952,A -85,B 0,C 180,E1 -15589.636,E2 -15589.636} C_VEL
LIN {X 0,Y 320.883,Z 409.242,A -85,B 0,C 180,E1 -15591.015,E2 -15591.015} C_VEL
LIN {X 0,Y 322.468,Z 397.443,A -85,B 0,C 180,E1 -15592.082,E2 -15592.082} C_VEL
LIN {X 0,Y 323.955,Z 385.178,A -85,B 0,C 180,E1 -15592.9,E2 -15592.9} C_VEL
LIN {X 0,Y 325.15,Z 372.415,A -85,B 0,C 180,E1 -15593.484,E2 -15593.484} C_VEL
LIN {X 0,Y 325.707,Z 357.455,A -85,B 0,C 180,E1 -15593.906,E2 -15593.906} C_VEL
LIN {X 0,Y 327.102,Z 303.645,A -85,B 0,C 180,E1 -15595.115,E2 -15595.115} C_VEL
LIN {X 0,Y 324.154,Z 281.927,A -85,B 0,C 180,E1 -15595.96,E2 -15595.96} C_VEL
LIN {X 0,Y 319.191,Z 253.806,A -85,B 0,C 180,E1 -15597.216,E2 -15597.216} C_VEL
LIN {X 0,Y 316.11,Z 245.471,A -85,B 0,C 180,E1 -15597.795,E2 -15597.795} C_VEL
LIN {X 0,Y 314.662,Z 240.997,A -85,B 0,C 180,E1 -15598.145,E2 -15598.145} C_VEL
LIN {X 0,Y 312.55,Z 230.548,A -85,B 0,C 180,E1 -15601.141,E2 -15601.141} C_VEL
LIN {X 0,Y 312.501,Z 230.523,A -85,B 0,C 180,E1 -15604.209,E2 -15604.209} C_VEL
LIN {X 0,Y 312.505,Z 230.559,A -85,B 0,C 180,E1 -15607.386,E2 -15607.386} C_VEL
LIN {X 0,Y 312.435,Z 230.566,A -85,B 0,C 180,E1 -15610.716,E2 -15610.716} C_VEL
LIN {X 0,Y 312.445,Z 230.557,A -85,B 0,C 180,E1 -15614.209,E2 -15614.209} C_VEL
LIN {X 0,Y 312.448,Z 230.548,A -85,B 0,C 180,E1 -15617.924,E2 -15617.924} C_VEL
LIN {X 0,Y 312.477,Z 230.557,A -85,B 0,C 180,E1 -15621.921,E2 -15621.921} C_VEL
LIN {X 0,Y 312.523,Z 230.531,A -85,B 0,C 180,E1 -15624.219,E2 -15624.219} C_VEL
LIN {X 0,Y 312.493,Z 230.557,A -85,B 0,C 180,E1 -15627.333,E2 -15627.333} C_VEL
LIN {X 0,Y 312.477,Z 230.534,A -85,B 0,C 180,E1 -15631.298,E2 -15631.298} C_VEL
LIN {X 0,Y 312.537,Z 230.55,A -85,B 0,C 180,E1 -15634.707,E2 -15634.707} C_VEL
LIN {X 0,Y 312.514,Z 230.527,A -85,B 0,C 180,E1 -15638.911,E2 -15638.911} C_VEL
LIN {X 0,Y 312.568,Z 230.544,A -85,B 0,C 180,E1 -15643.004,E2 -15643.004} C_VEL
LIN {X 0,Y 312.675,Z 230.504,A -85,B 0,C 180,E1 -15645.686,E2 -15645.686} C_VEL
LIN {X 0,Y 312.676,Z 230.534,A -85,B 0,C 180,E1 -15649.641,E2 -15649.641} C_VEL
LIN {X 0,Y 312.785,Z 230.512,A -85,B 0,C 180,E1 -15652.252,E2 -15652.252} C_VEL
LIN {X 0,Y 312.682,Z 230.504,A -85,B 0,C 180,E1 -15654.842,E2 -15654.842} C_VEL
LIN {X 0,Y 312.913,Z 230.499,A -85,B 0,C 180,E1 -15657.426,E2 -15657.426} C_VEL
LIN {X 0,Y 312.973,Z 230.479,A -85,B 0,C 180,E1 -15661.287,E2 -15661.287} C_VEL
LIN {X 0,Y 312.876,Z 230.506,A -85,B 0,C 180,E1 -15666.612,E2 -15666.612} C_VEL
LIN {X 0,Y 312.759,Z 230.507,A -85,B 0,C 180,E1 -15669.05,E2 -15669.05} C_VEL
LIN {X 0,Y 312.626,Z 230.535,A -85,B 0,C 180,E1 -15672.992,E2 -15672.992} C_VEL
LIN {X 0,Y 312.614,Z 230.533,A -85,B 0,C 180,E1 -15675.651,E2 -15675.651} C_VEL
LIN {X 0,Y 312.561,Z 230.546,A -85,B 0,C 180,E1 -15679.712,E2 -15679.712} C_VEL
LIN {X 0,Y 312.539,Z 230.541,A -85,B 0,C 180,E1 -15682.79,E2 -15682.79} C_VEL
LIN {X 0,Y 312.596,Z 230.546,A -85,B 0,C 180,E1 -15685.937,E2 -15685.937} C_VEL
LIN {X 0,Y 312.532,Z 230.541,A -85,B 0,C 180,E1 -15689.652,E2 -15689.652} C_VEL
LIN {X 0,Y 312.514,Z 230.546,A -85,B 0,C 180,E1 -15693.69,E2 -15693.69} C_VEL
LIN {X 0,Y 312.521,Z 230.553,A -85,B 0,C 180,E1 -15697.386,E2 -15697.386} C_VEL
LIN {X 0,Y 312.485,Z 230.564,A -85,B 0,C 180,E1 -15700.711,E2 -15700.711} C_VEL
LIN {X 0,Y 312.455,Z 230.563,A -85,B 0,C 180,E1 -15704.21,E2 -15704.21} C_VEL
LIN {X 0,Y 312.47,Z 230.558,A -85,B 0,C 180,E1 -15707.796,E2 -15707.796} C_VEL
LIN {X 0,Y 313.524,Z 233.448,A -85,B 0,C 180,E1 -15708.009,E2 -15708.009} C_VEL
LIN {X 0,Y 319.776,Z 244.281,A -85,B 0,C 180,E1 -15709.015,E2 -15709.015} C_VEL
LIN {X 0,Y 327.684,Z 259.946,A -85,B 0,C 180,E1 -15710.259,E2 -15710.259} C_VEL
LIN {X 0,Y 328.836,Z 262.971,A -85,B 0,C 180,E1 -15710.452,E2 -15710.452} C_VEL
LIN {X 0,Y 326.502,Z 339.826,A -85,B 0,C 180,E1 -15712.161,E2 -15712.161} C_VEL
LIN {X 0,Y 325.748,Z 353.318,A -85,B 0,C 180,E1 -15712.692,E2 -15712.692} C_VEL
LIN {X 0,Y 324.844,Z 364.762,A -85,B 0,C 180,E1 -15713.378,E2 -15713.378} C_VEL
LIN {X 0,Y 323.544,Z 376.168,A -85,B 0,C 180,E1 -15714.285,E2 -15714.285} C_VEL
LIN {X 0,Y 322.011,Z 387.296,A -85,B 0,C 180,E1 -15715.429,E2 -15715.429} C_VEL
LIN {X 0,Y 320.341,Z 397.46,A -85,B 0,C 180,E1 -15716.739,E2 -15716.739} C_VEL
LIN {X 0,Y 318.471,Z 407.61,A -85,B 0,C 180,E1 -15718.393,E2 -15718.393} C_VEL
LIN {X 0,Y 316.687,Z 416.785,A -85,B 0,C 180,E1 -15720.272,E2 -15720.272} C_VEL
LIN {X 0,Y 315.2,Z 423.826,A -85,B 0,C 180,E1 -15722.082,E2 -15722.082} C_VEL
LIN {X 0,Y 313.824,Z 430.144,A -85,B 0,C 180,E1 -15724.127,E2 -15724.127} C_VEL
LIN {X 0,Y 312.779,Z 434.991,A -85,B 0,C 180,E1 -15726.145,E2 -15726.145} C_VEL
LIN {X 0,Y 311.95,Z 438.663,A -85,B 0,C 180,E1 -15728.179,E2 -15728.179} C_VEL
LIN {X 0,Y 311.326,Z 441.238,A -85,B 0,C 180,E1 -15730.209,E2 -15730.209} C_VEL
LIN {X 0,Y 311.062,Z 442.431,A -85,B 0,C 180,E1 -15731.612,E2 -15731.612} C_VEL
LIN {X 0,Y 310.851,Z 443.094,A -85,B 0,C 180,E1 -15732.909,E2 -15732.909} C_VEL
LIN {X 0,Y 310.693,Z 443.386,A -85,B 0,C 180,E1 -15734.251,E2 -15734.251} C_VEL
LIN {X 0,Y 310.669,Z 442.894,A -85,B 0,C 180,E1 -15736.597,E2 -15736.597} C_VEL
LIN {X 0,Y 310.714,Z 441.728,A -85,B 0,C 180,E1 -15738.256,E2 -15738.256} C_VEL
LIN {X 0,Y 310.769,Z 440.361,A -85,B 0,C 180,E1 -15739.578,E2 -15739.578} C_VEL
LIN {X 0,Y 311.064,Z 437.453,A -85,B 0,C 180,E1 -15741.557,E2 -15741.557} C_VEL
LIN {X 0,Y 311.48,Z 433.5,A -85,B 0,C 180,E1 -15743.524,E2 -15743.524} C_VEL
LIN {X 0,Y 311.921,Z 428.402,A -85,B 0,C 180,E1 -15745.478,E2 -15745.478} C_VEL
LIN {X 0,Y 312.633,Z 421.964,A -85,B 0,C 180,E1 -15747.425,E2 -15747.425} C_VEL
LIN {X 0,Y 313.592,Z 413.959,A -85,B 0,C 180,E1 -15749.359,E2 -15749.359} C_VEL
LIN {X 0,Y 314.542,Z 405.787,A -85,B 0,C 180,E1 -15750.962,E2 -15750.962} C_VEL
LIN {X 0,Y 315.71,Z 395.73,A -85,B 0,C 180,E1 -15752.553,E2 -15752.553} C_VEL
LIN {X 0,Y 316.815,Z 385.813,A -85,B 0,C 180,E1 -15753.817,E2 -15753.817} C_VEL
LIN {X 0,Y 317.793,Z 375.264,A -85,B 0,C 180,E1 -15754.899,E2 -15754.899} C_VEL
LIN {X 0,Y 318.581,Z 363.318,A -85,B 0,C 180,E1 -15755.857,E2 -15755.857} C_VEL
LIN {X 0,Y 319.319,Z 350.362,A -85,B 0,C 180,E1 -15756.597,E2 -15756.597} C_VEL
LIN {X 0,Y 319.822,Z 336.619,A -85,B 0,C 180,E1 -15757.102,E2 -15757.102} C_VEL
LIN {X 0,Y 321.463,Z 258.399,A -85,B 0,C 180,E1 -15758.834,E2 -15758.834} C_VEL
LIN {X 0,Y 319.879,Z 249.284,A -85,B 0,C 180,E1 -15759.144,E2 -15759.144} C_VEL
LIN {X 0,Y 312.72,Z 230.531,A -85,B 0,C 180,E1 -15760.067,E2 -15760.067} C_VEL
LIN {X 0,Y 312.706,Z 230.532,A -85,B 0,C 180,E1 -15764.889,E2 -15764.889} C_VEL
LIN {X 0,Y 312.615,Z 230.542,A -85,B 0,C 180,E1 -15769.226,E2 -15769.226} C_VEL
LIN {X 0,Y 312.524,Z 230.553,A -85,B 0,C 180,E1 -15772.778,E2 -15772.778} C_VEL
LIN {X 0,Y 312.489,Z 230.557,A -85,B 0,C 180,E1 -15776.733,E2 -15776.733} C_VEL
LIN {X 0,Y 312.475,Z 230.562,A -85,B 0,C 180,E1 -15779.659,E2 -15779.659} C_VEL
LIN {X 0,Y 312.526,Z 230.557,A -85,B 0,C 180,E1 -15783.689,E2 -15783.689} C_VEL
LIN {X 0,Y 312.516,Z 230.555,A -85,B 0,C 180,E1 -15787.388,E2 -15787.388} C_VEL
LIN {X 0,Y 312.446,Z 230.562,A -85,B 0,C 180,E1 -15790.718,E2 -15790.718} C_VEL
LIN {X 0,Y 312.438,Z 230.559,A -85,B 0,C 180,E1 -15793.315,E2 -15793.315} C_VEL
LIN {X 0,Y 311.778,Z 230.645,A -85,B 0,C 180,E1 -15794.391,E2 -15794.391} C_VEL
LIN {X 0,Y 308.916,Z 231.002,A -85,B 0,C 180,E1 -15796.143,E2 -15796.143} C_VEL
LIN {X 0,Y 306.496,Z 231.306,A -85,B 0,C 180,E1 -15797.564,E2 -15797.564} C_VEL
LIN {X 0,Y 305.474,Z 231.431,A -85,B 0,C 180,E1 -15798.664,E2 -15798.664} C_VEL
LIN {X 0,Y 305.4,Z 231.439,A -85,B 0,C 180,E1 -15799.037,E2 -15799.037} C_VEL
LIN {X 0,Y 305.451,Z 231.431,A -85,B 0,C 180,E1 -15801.593,E2 -15801.593} C_VEL
LIN {X 0,Y 305.467,Z 231.434,A -85,B 0,C 180,E1 -15804.887,E2 -15804.887} C_VEL
LIN {X 0,Y 305.445,Z 231.434,A -85,B 0,C 180,E1 -15808.359,E2 -15808.359} C_VEL
LIN {X 0,Y 305.469,Z 231.427,A -85,B 0,C 180,E1 -15811.108,E2 -15811.108} C_VEL
LIN {X 0,Y 305.547,Z 231.487,A -85,B 0,C 180,E1 -15815.581,E2 -15815.581} C_VEL
LIN {X 0,Y 305.871,Z 233.171,A -85,B 0,C 180,E1 -15816.079,E2 -15816.079} C_VEL
LIN {X 0,Y 311.322,Z 254.007,A -85,B 0,C 180,E1 -15817.034,E2 -15817.034} C_VEL
LIN {X 0,Y 312.333,Z 259.901,A -85,B 0,C 180,E1 -15817.277,E2 -15817.277} C_VEL
LIN {X 0,Y 309.504,Z 341.709,A -85,B 0,C 180,E1 -15820.042,E2 -15820.042} C_VEL
LIN {X 0,Y 309.053,Z 355.111,A -85,B 0,C 180,E1 -15820.747,E2 -15820.747} C_VEL
LIN {X 0,Y 308.496,Z 366.684,A -85,B 0,C 180,E1 -15821.573,E2 -15821.573} C_VEL
LIN {X 0,Y 307.674,Z 379.112,A -85,B 0,C 180,E1 -15822.725,E2 -15822.725} C_VEL
LIN {X 0,Y 306.846,Z 390.47,A -85,B 0,C 180,E1 -15824.047,E2 -15824.047} C_VEL
LIN {X 0,Y 306.198,Z 400.871,A -85,B 0,C 180,E1 -15825.545,E2 -15825.545} C_VEL
LIN {X 0,Y 305.381,Z 411.159,A -85,B 0,C 180,E1 -15827.371,E2 -15827.371} C_VEL
LIN {X 0,Y 304.827,Z 418.842,A -85,B 0,C 180,E1 -15829.035,E2 -15829.035} C_VEL
LIN {X 0,Y 304.364,Z 426.35,A -85,B 0,C 180,E1 -15831.033,E2 -15831.033} C_VEL
LIN {X 0,Y 303.992,Z 433.219,A -85,B 0,C 180,E1 -15833.362,E2 -15833.362} C_VEL
LIN {X 0,Y 303.844,Z 437.726,A -85,B 0,C 180,E1 -15835.356,E2 -15835.356} C_VEL
LIN {X 0,Y 303.757,Z 441.08,A -85,B 0,C 180,E1 -15837.347,E2 -15837.347} C_VEL
LIN {X 0,Y 303.718,Z 442.712,A -85,B 0,C 180,E1 -15838.674,E2 -15838.674} C_VEL
LIN {X 0,Y 303.788,Z 443.902,A -85,B 0,C 180,E1 -15840,E2 -15840} C_VEL
LIN {X 0,Y 303.951,Z 444.68,A -85,B 0,C 180,E1 -15841.325,E2 -15841.325} C_VEL
LIN {X 0,Y 304.185,Z 445.022,A -85,B 0,C 180,E1 -15842.648,E2 -15842.648} C_VEL
LIN {X 0,Y 304.535,Z 444.901,A -85,B 0,C 180,E1 -15843.97,E2 -15843.97} C_VEL
LIN {X 0,Y 304.969,Z 444.372,A -85,B 0,C 180,E1 -15845.289,E2 -15845.289} C_VEL
LIN {X 0,Y 305.264,Z 443.455,A -85,B 0,C 180,E1 -15846.61,E2 -15846.61} C_VEL
LIN {X 0,Y 305.527,Z 442.11,A -85,B 0,C 180,E1 -15847.933,E2 -15847.933} C_VEL
LIN {X 0,Y 307.048,Z 438.633,A -85,B 0,C 180,E1 -15850.185,E2 -15850.185} C_VEL
LIN {X 0,Y 308.725,Z 433.648,A -85,B 0,C 180,E1 -15852.489,E2 -15852.489} C_VEL
LIN {X 0,Y 310.818,Z 427.052,A -85,B 0,C 180,E1 -15854.736,E2 -15854.736} C_VEL
LIN {X 0,Y 312.872,Z 419.919,A -85,B 0,C 180,E1 -15856.642,E2 -15856.642} C_VEL
LIN {X 0,Y 315.318,Z 411.125,A -85,B 0,C 180,E1 -15858.518,E2 -15858.518} C_VEL
LIN {X 0,Y 318.136,Z 400.118,A -85,B 0,C 180,E1 -15860.361,E2 -15860.361} C_VEL
LIN {X 0,Y 320.401,Z 389.985,A -85,B 0,C 180,E1 -15861.725,E2 -15861.725} C_VEL
LIN {X 0,Y 322.55,Z 379.032,A -85,B 0,C 180,E1 -15862.922,E2 -15862.922} C_VEL
LIN {X 0,Y 324.627,Z 367.097,A -85,B 0,C 180,E1 -15863.949,E2 -15863.949} C_VEL
LIN {X 0,Y 326.343,Z 354.24,A -85,B 0,C 180,E1 -15864.815,E2 -15864.815} C_VEL
LIN {X 0,Y 327.951,Z 339.415,A -85,B 0,C 180,E1 -15865.506,E2 -15865.506} C_VEL
LIN {X 0,Y 334.138,Z 281.464,A -85,B 0,C 180,E1 -15867.73,E2 -15867.73} C_VEL
LIN {X 0,Y 330.746,Z 274.449,A -85,B 0,C 180,E1 -15868.961,E2 -15868.961} C_VEL
LIN {X 0,Y 327.107,Z 267.996,A -85,B 0,C 180,E1 -15870.368,E2 -15870.368} C_VEL
